IF Main.Errors.InMoldDryingErrors.TopMoldB.HeatingZone[6].PT100_HasWrongPosition THEN 
Topmold_B_heating_Zone_6_PT100_wrong_position.Raise(0); 
END_IF 

IF Main.Errors.InMoldDryingErrors.TopMoldB.HeatingZone[6].PT100_Loose THEN 
Topmold_B_heating_Zone_6_PT100_loose.Raise(0); 
END_IF 

IF Main.Errors.InMoldDryingErrors.TopMoldB.HeatingZone[6].PT100_NotInserted THEN 
Topmold_B_heating_Zone_6_PT100_not_inserted.Raise(0); 
END_IF 

IF Main.Errors.InMoldDryingErrors.TopMoldB.HeatingZone[6].PT100_TempAboveSetpoint THEN 
Topmold_B_heating_Zone_6_Temperature_above_setpoint.Raise(0); 
END_IF 

IF Main.Errors.InMoldDryingErrors.TopMoldB.HeatingZone[6].PT100_TempBelowSetpoint THEN 
Topmold_B_heating_Zone_6_Temperature_below_setpoint.Raise(0); 
END_IF 

IF Main.Errors.InMoldDryingErrors.TopMoldB.HeatingZone[6].PT100_WireBreak THEN 
Topmold_B_heating_Zone_6_PT100_wirebreak.Raise(0); 
END_IF 

IF Main.Errors.InMoldDryingErrors.TopMoldB.HeatingZone[6].Thermal THEN 
Topmold_B_heating_Zone_6_Thermal.Raise(0); 
END_IF 

IF Main.Errors.InMoldDryingErrors.TopMoldB.HeatingZone[6].PT100_TemperatureAboveMaximum THEN 
Topmold_B_heating_zone_6_temperature_above_250_degree_heating_element_switched_off.Raise(0); 
END_IF 

IF Main.Errors.InMoldDryingErrors.TopMoldB.HeatingZone[6].PT100_TemperatureTooHighWarn THEN 
Topmold_B_heating_zone_6_temperature_above_230_degree.Raise(0); 
END_IF 

IF Main.Errors.InMoldDryingErrors.TopMoldB.Hydraulic.BallufError THEN 
Bottom_mold_B_error_on_balluf.Raise(0); 
END_IF 

IF Main.Errors.InMoldDryingErrors.TopMoldB.Hydraulic.IsMovingWithoutActivation THEN 
Bottom_mold_B_is_moving_without_activation.Raise(0); 
END_IF 

IF FALSE THEN 
Top_mold_B_Bot_side_pressure_too_high.Raise(0); 
END_IF 

IF FALSE THEN 
Top_mold_B_Rot_side_pressure_too_high.Raise(0); 
END_IF 

IF Main.Errors.InMoldDryingErrors.BottomMoldB.HeatingZone[1].PT100_ConnectorNotConnected THEN 
Bottom_mold_B_heating_Zone_1_connector_not_connected.Raise(0); 
END_IF 

IF Main.Errors.InMoldDryingErrors.BottomMoldB.HeatingZone[1].PT100_HasWrongPosition THEN 
Bottom_mold_B_heating_Zone_1_PT100_wrong_position.Raise(0); 
END_IF 

IF Main.Errors.InMoldDryingErrors.BottomMoldB.HeatingZone[1].PT100_Loose THEN 
Bottom_mold_B_heating_Zone_1_PT100_loose.Raise(0); 
END_IF 

IF Main.Errors.InMoldDryingErrors.BottomMoldB.HeatingZone[1].PT100_NotInserted THEN 
Bottom_mold_B_heating_Zone_1_PT100_not_inserted.Raise(0); 
END_IF 

IF Main.Errors.InMoldDryingErrors.BottomMoldB.HeatingZone[1].PT100_TempAboveSetpoint THEN 
Bottom_mold_B_heating_Zone_1_Temperature_above_setpoint.Raise(0); 
END_IF 

IF Main.Errors.InMoldDryingErrors.BottomMoldB.HeatingZone[1].PT100_TempBelowSetpoint THEN 
Bottom_mold_B_heating_Zone_1_Temperature_below_setpoint.Raise(0); 
END_IF 

IF Main.Errors.InMoldDryingErrors.BottomMoldB.HeatingZone[1].PT100_WireBreak THEN 
Bottom_mold_B_heating_Zone_1_PT100_wirebreak.Raise(0); 
END_IF 

IF Main.Errors.InMoldDryingErrors.BottomMoldB.HeatingZone[1].Thermal THEN 
Bottom_mold_B_heating_Zone_1_Thermal.Raise(0); 
END_IF 

IF Main.Errors.InMoldDryingErrors.BottomMoldB.HeatingZone[1].PT100_TemperatureAboveMaximum THEN 
Bottom_mold_B_heating_zone_1_temperature_above_250_degree_heating_element_switched_off.Raise(0); 
END_IF 

IF Main.Errors.InMoldDryingErrors.BottomMoldB.HeatingZone[1].PT100_TemperatureTooHighWarn THEN 
Bottom_mold_B_heating_zone_1_temperature_above_230_degree.Raise(0); 
END_IF 

IF Main.Errors.InMoldDryingErrors.BottomMoldB.HeatingZone[2].PT100_ConnectorNotConnected THEN 
Bottom_mold_B_heating_Zone_2_connector_not_connected.Raise(0); 
END_IF 

IF Main.Errors.InMoldDryingErrors.BottomMoldB.HeatingZone[2].PT100_HasWrongPosition THEN 
Bottom_mold_B_heating_Zone_2_PT100_wrong_position.Raise(0); 
END_IF 

IF Main.Errors.InMoldDryingErrors.BottomMoldB.HeatingZone[2].PT100_Loose THEN 
Bottom_mold_B_heating_Zone_2_PT100_loose.Raise(0); 
END_IF 

IF Main.Errors.InMoldDryingErrors.BottomMoldB.HeatingZone[2].PT100_NotInserted THEN 
Bottom_mold_B_heating_Zone_2_PT100_not_inserted.Raise(0); 
END_IF 

IF Main.Errors.InMoldDryingErrors.BottomMoldB.HeatingZone[2].PT100_TempAboveSetpoint THEN 
Bottom_mold_B_heating_Zone_2_Temperature_above_setpoint.Raise(0); 
END_IF 

IF Main.Errors.InMoldDryingErrors.BottomMoldB.HeatingZone[2].PT100_TempBelowSetpoint THEN 
Bottom_mold_B_heating_Zone_2_Temperature_below_setpoint.Raise(0); 
END_IF 

IF Main.Errors.InMoldDryingErrors.BottomMoldB.HeatingZone[2].PT100_WireBreak THEN 
Bottom_mold_B_heating_Zone_2_PT100_wirebreak.Raise(0); 
END_IF 

IF Main.Errors.InMoldDryingErrors.BottomMoldB.HeatingZone[2].Thermal THEN 
Bottom_mold_B_heating_Zone_2_Thermal.Raise(0); 
END_IF 

IF Main.Errors.InMoldDryingErrors.BottomMoldB.HeatingZone[2].PT100_TemperatureAboveMaximum THEN 
Bottom_mold_B_heating_zone_2_temperature_above_250_degree_heating_element_switched_off.Raise(0); 
END_IF 

IF Main.Errors.InMoldDryingErrors.BottomMoldB.HeatingZone[2].PT100_TemperatureTooHighWarn THEN 
Bottom_mold_B_heating_zone_2_temperature_above_230_degree.Raise(0); 
END_IF 

IF Main.Errors.InMoldDryingErrors.BottomMoldB.HeatingZone[3].PT100_ConnectorNotConnected THEN 
Bottom_mold_B_heating_Zone_3_connector_not_connected.Raise(0); 
END_IF 

IF Main.Errors.InMoldDryingErrors.BottomMoldB.HeatingZone[3].PT100_HasWrongPosition THEN 
Bottom_mold_B_heating_Zone_3_PT100_wrong_position.Raise(0); 
END_IF 

IF Main.Errors.InMoldDryingErrors.BottomMoldB.HeatingZone[3].PT100_Loose THEN 
Bottom_mold_B_heating_Zone_3_PT100_loose.Raise(0); 
END_IF 

IF Main.Errors.InMoldDryingErrors.BottomMoldB.HeatingZone[3].PT100_NotInserted THEN 
Bottom_mold_B_heating_Zone_3_PT100_not_inserted.Raise(0); 
END_IF 

IF Main.Errors.InMoldDryingErrors.BottomMoldB.HeatingZone[3].PT100_TempAboveSetpoint THEN 
Bottom_mold_B_heating_Zone_3_Temperature_above_setpoint.Raise(0); 
END_IF 

IF Main.Errors.InMoldDryingErrors.BottomMoldB.HeatingZone[3].PT100_TempBelowSetpoint THEN 
Bottom_mold_B_heating_Zone_3_Temperature_below_setpoint.Raise(0); 
END_IF 

IF Main.Errors.InMoldDryingErrors.BottomMoldB.HeatingZone[3].PT100_WireBreak THEN 
Bottom_mold_B_heating_Zone_3_PT100_wirebreak.Raise(0); 
END_IF 

IF Main.Errors.InMoldDryingErrors.BottomMoldB.HeatingZone[3].Thermal THEN 
Bottom_mold_B_heating_Zone_3_Thermal.Raise(0); 
END_IF 

IF Main.Errors.InMoldDryingErrors.BottomMoldB.HeatingZone[3].PT100_TemperatureAboveMaximum THEN 
Bottom_mold_B_heating_zone_3_temperature_above_250_degree_heating_element_switched_off.Raise(0); 
END_IF 

IF Main.Errors.InMoldDryingErrors.BottomMoldB.HeatingZone[3].PT100_TemperatureTooHighWarn THEN 
Bottom_mold_B_heating_zone_3_temperature_above_230_degree.Raise(0); 
END_IF 

IF Main.Errors.InMoldDryingErrors.BottomMoldB.HeatingZone[4].PT100_ConnectorNotConnected THEN 
Bottom_mold_B_heating_Zone_4_connector_not_connected.Raise(0); 
END_IF 

IF Main.Errors.InMoldDryingErrors.BottomMoldB.HeatingZone[4].PT100_HasWrongPosition THEN 
Bottom_mold_B_heating_Zone_4_PT100_wrong_position.Raise(0); 
END_IF 

IF Main.Errors.InMoldDryingErrors.BottomMoldB.HeatingZone[4].PT100_Loose THEN 
Bottom_mold_B_heating_Zone_4_PT100_loose.Raise(0); 
END_IF 

IF Main.Errors.InMoldDryingErrors.BottomMoldB.HeatingZone[4].PT100_NotInserted THEN 
Bottom_mold_B_heating_Zone_4_PT100_not_inserted.Raise(0); 
END_IF 

IF Main.Errors.InMoldDryingErrors.BottomMoldB.HeatingZone[4].PT100_TempAboveSetpoint THEN 
Bottom_mold_B_heating_Zone_4_Temperature_above_setpoint.Raise(0); 
END_IF 

IF Main.Errors.InMoldDryingErrors.BottomMoldB.HeatingZone[4].PT100_TempBelowSetpoint THEN 
Bottom_mold_B_heating_Zone_4_Temperature_below_setpoint.Raise(0); 
END_IF 

IF Main.Errors.InMoldDryingErrors.BottomMoldB.HeatingZone[4].PT100_WireBreak THEN 
Bottom_mold_B_heating_Zone_4_PT100_wirebreak.Raise(0); 
END_IF 

IF Main.Errors.InMoldDryingErrors.BottomMoldB.HeatingZone[4].Thermal THEN 
Bottom_mold_B_heating_Zone_4_Thermal.Raise(0); 
END_IF 

IF Main.Errors.InMoldDryingErrors.BottomMoldB.HeatingZone[4].PT100_TemperatureAboveMaximum THEN 
Bottom_mold_B_heating_zone_4_temperature_above_250_degree_heating_element_switched_off.Raise(0); 
END_IF 

IF Main.Errors.InMoldDryingErrors.BottomMoldB.HeatingZone[4].PT100_TemperatureTooHighWarn THEN 
Bottom_mold_B_heating_zone_4_temperature_above_230_degree.Raise(0); 
END_IF 

IF Main.Errors.InMoldDryingErrors.BottomMoldB.HeatingZone[5].PT100_ConnectorNotConnected THEN 
Bottom_mold_B_heating_Zone_5_connector_not_connected.Raise(0); 
END_IF 

IF Main.Errors.InMoldDryingErrors.BottomMoldB.HeatingZone[5].PT100_HasWrongPosition THEN 
Bottom_mold_B_heating_Zone_5_PT100_wrong_position.Raise(0); 
END_IF 

IF Main.Errors.InMoldDryingErrors.BottomMoldB.HeatingZone[5].PT100_Loose THEN 
Bottom_mold_B_heating_Zone_5_PT100_loose.Raise(0); 
END_IF 

IF Main.Errors.InMoldDryingErrors.BottomMoldB.HeatingZone[5].PT100_NotInserted THEN 
Bottom_mold_B_heating_Zone_5_PT100_not_inserted.Raise(0); 
END_IF 

IF Main.Errors.InMoldDryingErrors.BottomMoldB.HeatingZone[5].PT100_TempAboveSetpoint THEN 
Bottom_mold_B_heating_Zone_5_Temperature_above_setpoint.Raise(0); 
END_IF 

IF Main.Errors.InMoldDryingErrors.BottomMoldB.HeatingZone[5].PT100_TempBelowSetpoint THEN 
Bottom_mold_B_heating_Zone_5_Temperature_below_setpoint.Raise(0); 
END_IF 

IF Main.Errors.InMoldDryingErrors.BottomMoldB.HeatingZone[5].PT100_WireBreak THEN 
Bottom_mold_B_heating_Zone_5_PT100_wirebreak.Raise(0); 
END_IF 

IF Main.Errors.InMoldDryingErrors.BottomMoldB.HeatingZone[5].Thermal THEN 
Bottom_mold_B_heating_Zone_5_Thermal.Raise(0); 
END_IF 

IF Main.Errors.InMoldDryingErrors.BottomMoldB.HeatingZone[5].PT100_TemperatureAboveMaximum THEN 
Bottom_mold_B_heating_zone_5_temperature_above_250_degree_heating_element_switched_off.Raise(0); 
END_IF 

IF Main.Errors.InMoldDryingErrors.BottomMoldB.HeatingZone[5].PT100_TemperatureTooHighWarn THEN 
Bottom_mold_B_heating_zone_5_temperature_above_230_degree.Raise(0); 
END_IF 

IF Main.Errors.InMoldDryingErrors.BottomMoldB.HeatingZone[6].PT100_ConnectorNotConnected THEN 
Bottom_mold_B_heating_Zone_6_connector_not_connected.Raise(0); 
END_IF 

IF Main.Errors.InMoldDryingErrors.BottomMoldB.HeatingZone[6].PT100_HasWrongPosition THEN 
Bottom_mold_B_heating_Zone_6_PT100_wrong_position.Raise(0); 
END_IF 

IF Main.Errors.InMoldDryingErrors.BottomMoldB.HeatingZone[6].PT100_Loose THEN 
Bottom_mold_B_heating_Zone_6_PT100_loose.Raise(0); 
END_IF 

IF Main.Errors.InMoldDryingErrors.BottomMoldB.HeatingZone[6].PT100_NotInserted THEN 
Bottom_mold_B_heating_Zone_6_PT100_not_inserted.Raise(0); 
END_IF 

IF Main.Errors.InMoldDryingErrors.BottomMoldB.HeatingZone[6].PT100_TempAboveSetpoint THEN 
Bottom_mold_B_heating_Zone_6_Temperature_above_setpoint.Raise(0); 
END_IF 

IF Main.Errors.InMoldDryingErrors.BottomMoldB.HeatingZone[6].PT100_TempBelowSetpoint THEN 
Bottom_mold_B_heating_Zone_6_Temperature_below_setpoint.Raise(0); 
END_IF 

IF Main.Errors.InMoldDryingErrors.BottomMoldB.HeatingZone[6].PT100_WireBreak THEN 
Bottom_mold_B_heating_Zone_6_PT100_wirebreak.Raise(0); 
END_IF 

IF Main.Errors.InMoldDryingErrors.BottomMoldB.HeatingZone[6].Thermal THEN 
Bottom_mold_B_heating_Zone_6_Thermal.Raise(0); 
END_IF 

IF Main.Errors.InMoldDryingErrors.BottomMoldB.HeatingZone[6].PT100_TemperatureAboveMaximum THEN 
Bottom_mold_B_heating_zone_6_temperature_above_250_degree_heating_element_switched_off.Raise(0); 
END_IF 

IF Main.Errors.InMoldDryingErrors.BottomMoldB.HeatingZone[6].PT100_TemperatureTooHighWarn THEN 
Bottom_mold_B_heating_zone_6_temperature_above_230_degree.Raise(0); 
END_IF 

IF Main.Errors.InMoldDryingErrors.BottomMoldA.HorizontalCilinder.Cilinder THEN 
Takeout_unit_A_horizontal_cylinder_error.Raise(0); 
END_IF 

IF Main.Errors.InMoldDryingErrors.BottomMoldA.HorizontalCilinder.CilinderSlow_IN THEN 
Takeout_unit_A_horizontal_cylinder_timeout_in.Raise(0); 
END_IF 

IF Main.Errors.InMoldDryingErrors.BottomMoldA.HorizontalCilinder.CilinderSlow_OUT THEN 
Takeout_unit_A_horizontal_cylinder_timeout_out.Raise(0); 
END_IF 

IF Main.Errors.InMoldDryingErrors.BottomMoldB.HorizontalCilinder.Cilinder THEN 
Takeout_unit_B_horizontal_cylinder_error.Raise(0); 
END_IF 

IF Main.Errors.InMoldDryingErrors.BottomMoldB.HorizontalCilinder.CilinderSlow_IN THEN 
Takeout_unit_B_horizontal_cylinder_timeout_in.Raise(0); 
END_IF 

IF Main.Errors.InMoldDryingErrors.BottomMoldB.HorizontalCilinder.CilinderSlow_OUT THEN 
Takeout_unit_B_horizontal_cylinder_timeout_out.Raise(0); 
END_IF 

IF Main.Errors.InMoldDryingErrors.BottomMoldA.VerticalCilinder.Cilinder THEN 
Takeout_unit_A_vertical_cylinder_error.Raise(0); 
END_IF 

IF Main.Errors.InMoldDryingErrors.BottomMoldA.VerticalCilinder.CilinderSlow_IN THEN 
Takeout_unit_A_vertical_cylinder_timeout_in.Raise(0); 
END_IF 

IF Main.Errors.InMoldDryingErrors.BottomMoldA.VerticalCilinder.CilinderSlow_OUT THEN 
Takeout_unit_A_vertical_cylinder_timeout_out.Raise(0); 
END_IF 

IF Main.Errors.InMoldDryingErrors.BottomMoldB.VerticalCilinder.Cilinder THEN 
Takeout_unit_B_vertical_cylinder_error.Raise(0); 
END_IF 

IF Main.Errors.InMoldDryingErrors.BottomMoldB.VerticalCilinder.CilinderSlow_IN THEN 
Takeout_unit_B_vertical_cylinder_timeout_in.Raise(0); 
END_IF 

IF Main.Errors.InMoldDryingErrors.BottomMoldB.VerticalCilinder.CilinderSlow_OUT THEN 
Takeout_unit_B_vertical_cylinder_timeout_out.Raise(0); 
END_IF 

IF Main.Errors.InMoldDryingErrors.BottomMoldA.VacuumSection[1] THEN 
Takeout_unit_A_error_on_vacuum_section_1.Raise(0); 
END_IF 

IF Main.Errors.InMoldDryingErrors.BottomMoldA.VacuumSection[2] THEN 
Takeout_unit_A_error_on_vacuum_section_2.Raise(0); 
END_IF 

IF Main.Errors.InMoldDryingErrors.BottomMoldA.VacuumSection[3] THEN 
Takeout_unit_A_error_on_vacuum_section_3.Raise(0); 
END_IF 

IF Main.Errors.InMoldDryingErrors.BottomMoldA.VacuumSection[4] THEN 
Takeout_unit_A_error_on_vacuum_section_4.Raise(0); 
END_IF 

IF Main.Errors.InMoldDryingErrors.BottomMoldB.VacuumSection[1] THEN 
Takeout_unit_B_error_on_vacuum_section_1.Raise(0); 
END_IF 

IF Main.Errors.InMoldDryingErrors.BottomMoldB.VacuumSection[2] THEN 
Takeout_unit_B_error_on_vacuum_section_2.Raise(0); 
END_IF 

IF Main.Errors.InMoldDryingErrors.BottomMoldB.VacuumSection[3] THEN 
Takeout_unit_B_error_on_vacuum_section_3.Raise(0); 
END_IF 

IF Main.Errors.InMoldDryingErrors.BottomMoldB.VacuumSection[4] THEN 
Takeout_unit_B_error_on_vacuum_section_4.Raise(0); 
END_IF 

IF Main.Errors.InMoldDryingErrors.ProductForming.HydraulicPump.Maintenance THEN 
Machine_pond_hydraulic_pump_maintenance_switch.Raise(0); 
END_IF 

IF Main.Errors.InMoldDryingErrors.ProductForming.HydraulicPump.Thermal THEN 
Machine_pond_hydraulic_pump_thermal_error.Raise(0); 
END_IF 

IF Main.Errors.InMoldDryingErrors.ProductForming.MachinePond.FeedingPulp.Cilinder THEN 
Machine_oond_pulp_feeding_cylinder_error.Raise(0); 
END_IF 

IF Main.Errors.InMoldDryingErrors.ProductForming.MachinePond.FeedingPulp.CilinderSlow_IN THEN 
Machine_pond_pulp_feeding_cylinder_timeout_in.Raise(0); 
END_IF 

IF Main.Errors.InMoldDryingErrors.ProductForming.MachinePond.FeedingPulp.CilinderSlow_OUT THEN 
Machine_pond_pulp_feeding_cylinder_timeout_out.Raise(0); 
END_IF 

IF Main.Errors.InMoldDryingErrors.TransferMold.HydraulicCilinder.BallufError THEN 
Transfermold_error_on_balluf.Raise(0); 
END_IF 

IF Main.Errors.InMoldDryingErrors.TransferMold.HydraulicCilinder.IsMovingWithoutActivation THEN 
Transfermold_is_moving_without_activation.Raise(0); 
END_IF 

IF Main.Errors.InMoldDryingErrors.RH_BotMoldAToCoolForTrMDown THEN 
RHSR_Bottommold_A_too_cool_for_transfermold_to_come_down.Raise(0); 
END_IF 

IF Main.Errors.InMoldDryingErrors.RH_BotMoldBToCoolForTrMDown THEN 
RHSR_Bottommold_B_too_cool_for_transfermold_to_come_down.Raise(0); 
END_IF 

IF Main.Errors.ProductHandlingErrors.Gantry_A.Collision THEN 
Gantry_A_collision_detected.Raise(0); 
END_IF 

IF Main.Errors.ProductHandlingErrors.Gantry_A.EndLimitHorBack THEN 
Gantry_A_Horizontal_limit_endswitch_backside.Raise(0); 
END_IF 

IF Main.Errors.ProductHandlingErrors.Gantry_A.EndLimitHorFront THEN 
Gantry_A_Horizontal_limit_endswitch_frontside.Raise(0); 
END_IF 

IF Main.Errors.ProductHandlingErrors.Gantry_A.EndLimitVertDown THEN 
Gantry_A_vertical_limit_endswitch_down.Raise(0); 
END_IF 

IF Main.Errors.ProductHandlingErrors.Gantry_A.EndLimitVertUp THEN 
Gantry_A_vertical_limit_endswitch_up.Raise(0); 
END_IF 

IF Main.Errors.ProductHandlingErrors.Gantry_A.HorizontalNCAxisError.exDriveAbsoluut THEN 
Gantry_A_Horizontal_Drive_absoluut_error.Raise(0); 
END_IF 

IF Main.Errors.ProductHandlingErrors.Gantry_A.HorizontalNCAxisError.exDriveJog THEN 
Gantry_A_Horizontal_Drive_Jog_error.Raise(0); 
END_IF 

IF Main.Errors.ProductHandlingErrors.Gantry_A.HorizontalNCAxisError.exDrivePower THEN 
Gantry_A_Horizontal_Drive_power_error.Raise(0); 
END_IF 

IF Main.Errors.ProductHandlingErrors.Gantry_A.HorizontalNCAxisError.exDriveReset THEN 
Gantry_A_Horizontal_Drive_reset.Raise(0); 
END_IF 

IF Main.Errors.ProductHandlingErrors.Gantry_A.HorizontalNCAxisError.exDriveStatus THEN 
Gantry_A_Horizontal_Drive_status.Raise(0); 
END_IF 

IF Main.Errors.ProductHandlingErrors.Gantry_A.HorizontalNCAxisError.exDriveStop THEN 
Gantry_A_Horizontal_Drive_stop_error.Raise(0); 
END_IF 

IF Main.Errors.ProductHandlingErrors.Gantry_A.HorizontalNCAxisError.exDriveVelocity THEN 
Gantry_A_Horizontal_Drive_velocity_error.Raise(0); 
END_IF 

IF Main.Errors.ProductHandlingErrors.Gantry_A.HorizontalNCAxisError.exHome THEN 
Gantry_A_Horizontal_Drive_home_error.Raise(0); 
END_IF 

IF Main.Errors.ProductHandlingErrors.Gantry_A.HorizontalNCAxisError.exLagError THEN 
Gantry_A_Horizontal_Drive_lag_error.Raise(0); 
END_IF 

IF Main.Errors.ProductHandlingErrors.Gantry_A.HorizontalNCAxisError.exReadParameter THEN 
Gantry_A_Horizontal_Drive_read_parameter_error.Raise(0); 
END_IF 

IF Main.Errors.ProductHandlingErrors.Gantry_A.HorizontalNCAxisError.exWriteParameter THEN 
Gantry_A_Horizontal_Drive_write_parameter_error.Raise(0); 
END_IF 

IF Main.Errors.ProductHandlingErrors.Gantry_B.Collision THEN 
Gantry_B_collision_detected.Raise(0); 
END_IF 

IF Main.Errors.ProductHandlingErrors.Gantry_B.EndLimitHorBack THEN 
Gantry_B_horizontal_limit_endswitch_backside.Raise(0); 
END_IF 

IF Main.Errors.ProductHandlingErrors.Gantry_B.EndLimitHorFront THEN 
Gantry_B_horizontal_limit_endswitch_frontside.Raise(0); 
END_IF 

IF Main.Errors.ProductHandlingErrors.Gantry_B.EndLimitVertDown THEN 
Gantry_B_vertical_limit_endswitch_down.Raise(0); 
END_IF 

IF Main.Errors.ProductHandlingErrors.Gantry_B.EndLimitVertUp THEN 
Gantry_B_vertical_limit_endswitch_up.Raise(0); 
END_IF 

IF Main.Errors.ProductHandlingErrors.Gantry_B.HorizontalNCAxisError.exDriveAbsoluut THEN 
Gantry_B_Horizontal_Drive_absoluut_error.Raise(0); 
END_IF 

IF Main.Errors.ProductHandlingErrors.Gantry_B.HorizontalNCAxisError.exDriveJog THEN 
Gantry_B_Horizontal_Drive_Jog_error.Raise(0); 
END_IF 

IF Main.Errors.ProductHandlingErrors.Gantry_B.HorizontalNCAxisError.exDrivePower THEN 
Gantry_B_Horizontal_Drive_power_error.Raise(0); 
END_IF 

IF Main.Errors.ProductHandlingErrors.Gantry_B.HorizontalNCAxisError.exDriveReset THEN 
Gantry_B_Horizontal_Drive_reset.Raise(0); 
END_IF 

IF Main.Errors.ProductHandlingErrors.Gantry_B.HorizontalNCAxisError.exDriveStatus THEN 
Gantry_B_Horizontal_Drive_status.Raise(0); 
END_IF 

IF Main.Errors.ProductHandlingErrors.Gantry_B.HorizontalNCAxisError.exDriveStop THEN 
Gantry_B_Horizontal_Drive_stop_error.Raise(0); 
END_IF 

IF Main.Errors.ProductHandlingErrors.Gantry_B.HorizontalNCAxisError.exDriveVelocity THEN 
Gantry_B_Horizontal_Drive_velocity_error.Raise(0); 
END_IF 

IF Main.Errors.ProductHandlingErrors.Gantry_B.HorizontalNCAxisError.exHome THEN 
Gantry_B_Horizontal_Drive_home_error.Raise(0); 
END_IF 

IF Main.Errors.ProductHandlingErrors.Gantry_B.HorizontalNCAxisError.exLagError THEN 
Gantry_B_Horizontal_Drive_lag_error.Raise(0); 
END_IF 

IF Main.Errors.ProductHandlingErrors.Gantry_B.HorizontalNCAxisError.exReadParameter THEN 
Gantry_B_Horizontal_Drive_read_parameter_error.Raise(0); 
END_IF 

IF Main.Errors.ProductHandlingErrors.Gantry_B.HorizontalNCAxisError.exWriteParameter THEN 
Gantry_B_Horizontal_Drive_write_parameter_error.Raise(0); 
END_IF 

IF Main.Errors.ProductHandlingErrors.RH_HorMovingVertNotAtTranspPos_A THEN 
RHSR_product_handling_gantry_A_is_moving_horizotal_while_vertical_not_on_position.Raise(0); 
END_IF 

IF Main.Errors.ProductHandlingErrors.RH_HorMovingVertNotAtTranspPos_B THEN 
RHSR_product_handling_gantry_B_is_moving_horizotal_while_vertical_not_on_position.Raise(0); 
END_IF 

IF Main.Errors.ProductHandlingErrors.RH_VertMovingHorNotInPos_A THEN 
RHSR_product_handling_gantry_A_is_moving_vertical_while_horizontal_not_on_position.Raise(0); 
END_IF 

IF Main.Errors.ProductHandlingErrors.RH_VertMovingHorNotInPos_B THEN 
RHSR_product_handling_gantry_B_is_moving_vertical_while_horizontal_not_on_position.Raise(0); 
END_IF 

IF Main.Errors.InMoldDryingErrors.ProductForming.SprayBar.NCAxisError.exDriveAbsoluut THEN 
Spraybar_Drive_absoluut_error.Raise(0); 
END_IF 

IF Main.Errors.InMoldDryingErrors.ProductForming.SprayBar.NCAxisError.exDriveJog THEN 
Spraybar_Drive_Jog_error.Raise(0); 
END_IF 

IF Main.Errors.InMoldDryingErrors.ProductForming.SprayBar.NCAxisError.exDrivePower THEN 
Spraybar_Drive_power_error.Raise(0); 
END_IF 

IF Main.Errors.InMoldDryingErrors.ProductForming.SprayBar.NCAxisError.exDriveReset THEN 
Spraybar_Drive_reset.Raise(0); 
END_IF 

IF Main.Errors.InMoldDryingErrors.ProductForming.SprayBar.NCAxisError.exDriveStatus THEN 
Spraybar_Drive_status.Raise(0); 
END_IF 

IF Main.Errors.InMoldDryingErrors.ProductForming.SprayBar.NCAxisError.exDriveStop THEN 
Spraybar_Drive_stop_error.Raise(0); 
END_IF 

IF Main.Errors.InMoldDryingErrors.ProductForming.SprayBar.NCAxisError.exDriveVelocity THEN 
Spraybar_Drive_velocity_error.Raise(0); 
END_IF 

IF Main.Errors.InMoldDryingErrors.ProductForming.SprayBar.NCAxisError.exHome THEN 
Spraybar_Drive_home_error.Raise(0); 
END_IF 

IF Main.Errors.InMoldDryingErrors.ProductForming.SprayBar.NCAxisError.exLagError THEN 
Spraybar_Drive_lag_error.Raise(0); 
END_IF 

IF Main.Errors.InMoldDryingErrors.ProductForming.SprayBar.NCAxisError.exReadParameter THEN 
Spraybar_Drive_read_parameter_error.Raise(0); 
END_IF 

IF Main.Errors.InMoldDryingErrors.ProductForming.SprayBar.NCAxisError.exWriteParameter THEN 
Spraybar_Drive_write_parameter_error.Raise(0); 
END_IF 

IF Main.Errors.ProductHandlingErrors.Gantry_A.ProductLost[1] THEN 
Gantry_A_product_lost_section_1.Raise(0); 
END_IF 

IF Main.Errors.ProductHandlingErrors.Gantry_A.ProductLost[2] THEN 
Gantry_A_product_lost_section_2.Raise(0); 
END_IF 

IF Main.Errors.ProductHandlingErrors.Gantry_A.ProductLost[3] THEN 
Gantry_A_product_lost_section_3.Raise(0); 
END_IF 

IF Main.Errors.ProductHandlingErrors.Gantry_A.ProductLost[4] THEN 
Gantry_A_product_lost_section_4.Raise(0); 
END_IF 

IF Main.Errors.ProductHandlingErrors.Gantry_A.ProductLost[5] THEN 
Gantry_A_product_lost_section_5.Raise(0); 
END_IF 

IF Main.Errors.ProductHandlingErrors.Gantry_A.ProductLost[6] THEN 
Gantry_A_product_lost_section_6.Raise(0); 
END_IF 

IF Main.Errors.ProductHandlingErrors.Gantry_B.ProductLost[1] THEN 
Gantry_B_product_lost_section_1.Raise(0); 
END_IF 

IF Main.Errors.ProductHandlingErrors.Gantry_B.ProductLost[2] THEN 
Gantry_B_product_lost_section_2.Raise(0); 
END_IF 

IF Main.Errors.ProductHandlingErrors.Gantry_B.ProductLost[3] THEN 
Gantry_B_product_lost_section_3.Raise(0); 
END_IF 

IF Main.Errors.ProductHandlingErrors.Gantry_B.ProductLost[4] THEN 
Gantry_B_product_lost_section_4.Raise(0); 
END_IF 

IF Main.Errors.ProductHandlingErrors.Gantry_B.ProductLost[5] THEN 
Gantry_B_product_lost_section_5.Raise(0); 
END_IF 

IF Main.Errors.ProductHandlingErrors.Gantry_B.ProductLost[6] THEN 
Gantry_B_product_lost_section_6.Raise(0); 
END_IF 

IF Main.Errors.InMoldDryingErrors.ProductForming.SprayBar.PositionAtFrontError THEN 
Spraybar_not_in_front_rest_position.Raise(0); 
END_IF 

IF Main.Errors.InMoldDryingErrors.ProductForming.SprayBar.PositionAtBackError THEN 
Spraybar_not_in_back_rest_position.Raise(0); 
END_IF 

IF MAIN.EtherCatDiag.EtherCATLinkError THEN 
Ethercat_diagnosed_a_link_error.Raise(0); 
END_IF 

IF MAIN.EtherCatDiag.EtherCATSlaveMissing THEN 
Ethercat_diagnosed_that_a_slave_is_missing.Raise(0); 
END_IF 

IF MAIN.EtherCatDiag.EtherCATOPmode THEN 
Ethercat_diagnosed_a_non_OP_state.Raise(0); 
END_IF 

IF MAIN.EtherCatDiag.EtherCATResetNeeded THEN 
Ethercat_diagnosed_that_a_ethercat_reset_is_needed.Raise(0); 
END_IF 

IF Main.Errors.InMoldDryingErrors.TopMoldA.Hydraulic.SafePositionValveNotReached THEN 
TopMold_A_Safe_position_not_reached.Raise(0); 
END_IF 

IF Main.Errors.InMoldDryingErrors.TopMoldB.Hydraulic.SafePositionValveNotReached THEN 
TopMold_B_Safe_position_not_reached.Raise(0); 
END_IF 

IF Main.Errors.InMoldDryingErrors.TransferMold.HydraulicCilinder.SafePositionValveNotReached THEN 
Transfermold_Safe_position_not_reached.Raise(0); 
END_IF 

IF Main.Errors.InMoldDryingErrors.TempDeviationToHighA[1] THEN 
Difference_in_temperature_too_high_top_bottommold_A_zone_1.Raise(0); 
END_IF 

IF Main.Errors.InMoldDryingErrors.TempDeviationToHighA[2] THEN 
Difference_in_temperature_too_high_top_bottommold_A_zone_2.Raise(0); 
END_IF 

IF Main.Errors.InMoldDryingErrors.TempDeviationToHighA[3] THEN 
Difference_in_temperature_too_high_top_bottommold_A_zone_3.Raise(0); 
END_IF 

IF Main.Errors.InMoldDryingErrors.TempDeviationToHighA[4] THEN 
Difference_in_temperature_too_high_top_bottommold_A_zone_4.Raise(0); 
END_IF 

IF Main.Errors.InMoldDryingErrors.TempDeviationToHighA[5] THEN 
Difference_in_temperature_too_high_top_bottommold_A_zone_5.Raise(0); 
END_IF 

IF Main.Errors.InMoldDryingErrors.TempDeviationToHighA[6] THEN 
Difference_in_temperature_too_high_top_bottommold_A_zone_6.Raise(0); 
END_IF 

IF Main.Errors.InMoldDryingErrors.TempDeviationToHighB[1] THEN 
Difference_in_temperature_too_high_top_bottommold_B_zone_1.Raise(0); 
END_IF 

IF Main.Errors.InMoldDryingErrors.TempDeviationToHighB[2] THEN 
Difference_in_temperature_too_high_top_bottommold_B_zone_2.Raise(0); 
END_IF 

IF Main.Errors.InMoldDryingErrors.TempDeviationToHighB[3] THEN 
Difference_in_temperature_too_high_top_bottommold_B_zone_3.Raise(0); 
END_IF 

IF Main.Errors.InMoldDryingErrors.TempDeviationToHighB[4] THEN 
Difference_in_temperature_too_high_top_bottommold_B_zone_4.Raise(0); 
END_IF 

IF Main.Errors.InMoldDryingErrors.TempDeviationToHighB[5] THEN 
Difference_in_temperature_too_high_top_bottommold_B_zone_5.Raise(0); 
END_IF 

IF Main.Errors.InMoldDryingErrors.TempDeviationToHighB[6] THEN 
Difference_in_temperature_too_high_top_bottommold_B_zone_6.Raise(0); 
END_IF 

IF Main.Errors.ProductHandlingErrors.Gantry_A.VerticalNCAxisError.exDriveAbsoluut THEN 
Gantry_A_Vertical_Drive_absoluut_error.Raise(0); 
END_IF 

IF Main.Errors.ProductHandlingErrors.Gantry_A.VerticalNCAxisError.exDriveJog THEN 
Gantry_A_Vertical_Drive_Jog_error.Raise(0); 
END_IF 

IF Main.Errors.ProductHandlingErrors.Gantry_A.VerticalNCAxisError.exDrivePower THEN 
Gantry_A_Vertical_Drive_power_error.Raise(0); 
END_IF 

IF Main.Errors.ProductHandlingErrors.Gantry_A.VerticalNCAxisError.exDriveReset THEN 
Gantry_A_Vertical_Drive_reset.Raise(0); 
END_IF 

IF Main.Errors.ProductHandlingErrors.Gantry_A.VerticalNCAxisError.exDriveStatus THEN 
Gantry_A_Vertical_Drive_status.Raise(0); 
END_IF 

IF Main.Errors.ProductHandlingErrors.Gantry_A.VerticalNCAxisError.exDriveStop THEN 
Gantry_A_Vertical_Drive_stop_error.Raise(0); 
END_IF 

IF Main.Errors.ProductHandlingErrors.Gantry_A.VerticalNCAxisError.exDriveVelocity THEN 
Gantry_A_Vertical_Drive_velocity_error.Raise(0); 
END_IF 

IF Main.Errors.ProductHandlingErrors.Gantry_A.VerticalNCAxisError.exHome THEN 
Gantry_A_Vertical_Drive_home_error.Raise(0); 
END_IF 

IF Main.Errors.ProductHandlingErrors.Gantry_A.VerticalNCAxisError.exLagError THEN 
Gantry_A_Vertical_Drive_lag_error.Raise(0); 
END_IF 

IF Main.Errors.ProductHandlingErrors.Gantry_A.VerticalNCAxisError.exReadParameter THEN 
Gantry_A_Vertical_Drive_read_parameter_error.Raise(0); 
END_IF 

IF Main.Errors.ProductHandlingErrors.Gantry_A.VerticalNCAxisError.exWriteParameter THEN 
Gantry_A_Vertical_Drive_write_parameter_error.Raise(0); 
END_IF 

IF Main.Errors.ProductHandlingErrors.Gantry_B.VerticalNCAxisError.exDriveAbsoluut THEN 
Gantry_B_Vertical_Drive_absoluut_error.Raise(0); 
END_IF 

IF Main.Errors.ProductHandlingErrors.Gantry_B.VerticalNCAxisError.exDriveJog THEN 
Gantry_B_Vertical_Drive_Jog_error.Raise(0); 
END_IF 

IF Main.Errors.ProductHandlingErrors.Gantry_B.VerticalNCAxisError.exDrivePower THEN 
Gantry_B_Vertical_Drive_power_error.Raise(0); 
END_IF 

IF Main.Errors.ProductHandlingErrors.Gantry_B.VerticalNCAxisError.exDriveReset THEN 
Gantry_B_Vertical_Drive_reset.Raise(0); 
END_IF 

IF Main.Errors.ProductHandlingErrors.Gantry_B.VerticalNCAxisError.exDriveStatus THEN 
Gantry_B_Vertical_Drive_status.Raise(0); 
END_IF 

IF Main.Errors.ProductHandlingErrors.Gantry_B.VerticalNCAxisError.exDriveStop THEN 
Gantry_B_Vertical_Drive_stop_error.Raise(0); 
END_IF 

IF Main.Errors.ProductHandlingErrors.Gantry_B.VerticalNCAxisError.exDriveVelocity THEN 
Gantry_B_Vertical_Drive_velocity_error.Raise(0); 
END_IF 

IF Main.Errors.ProductHandlingErrors.Gantry_B.VerticalNCAxisError.exHome THEN 
Gantry_B_Vertical_Drive_home_error.Raise(0); 
END_IF 

IF Main.Errors.ProductHandlingErrors.Gantry_B.VerticalNCAxisError.exLagError THEN 
Gantry_B_Vertical_Drive_lag_error.Raise(0); 
END_IF 

IF Main.Errors.ProductHandlingErrors.Gantry_B.VerticalNCAxisError.exReadParameter THEN 
Gantry_B_Vertical_Drive_read_parameter_error.Raise(0); 
END_IF 

IF Main.Errors.ProductHandlingErrors.Gantry_B.VerticalNCAxisError.exWriteParameter THEN 
Gantry_B_Vertical_Drive_write_parameter_error.Raise(0); 
END_IF 

IF Main.Errors.InMoldDryingErrors.BottomMoldB.HorizontalAxis.exDriveAbsoluut THEN 
Bottommold_B_Horizontal_Drive_absoluut_error.Raise(0); 
END_IF 

IF Main.Errors.InMoldDryingErrors.BottomMoldB.HorizontalAxis.exDriveJog THEN 
Bottommold_B_Horizontal_Drive_Jog_error.Raise(0); 
END_IF 

IF Main.Errors.InMoldDryingErrors.BottomMoldB.HorizontalAxis.exDrivePower THEN 
Bottommold_B_Horizontal_Drive_power_error.Raise(0); 
END_IF 

IF Main.Errors.InMoldDryingErrors.BottomMoldB.HorizontalAxis.exDriveReset THEN 
Bottommold_B_Horizontal_Drive_reset.Raise(0); 
END_IF 

IF Main.Errors.InMoldDryingErrors.BottomMoldB.HorizontalAxis.exDriveStatus THEN 
Bottommold_B_Horizontal_Drive_status.Raise(0); 
END_IF 

IF Main.Errors.InMoldDryingErrors.BottomMoldB.HorizontalAxis.exDriveStop THEN 
Bottommold_B_Horizontal_Drive_stop_error.Raise(0); 
END_IF 

IF Main.Errors.InMoldDryingErrors.BottomMoldB.HorizontalAxis.exDriveVelocity THEN 
Bottommold_B_Horizontal_Drive_velocity_error.Raise(0); 
END_IF 

IF Main.Errors.InMoldDryingErrors.BottomMoldB.HorizontalAxis.exHome THEN 
Bottommold_B_Horizontal_Drive_home_error.Raise(0); 
END_IF 

IF Main.Errors.InMoldDryingErrors.BottomMoldB.HorizontalAxis.exLagError THEN 
Bottommold_B_Horizontal_Drive_lag_error.Raise(0); 
END_IF 

IF Main.Errors.InMoldDryingErrors.BottomMoldB.HorizontalAxis.exReadParameter THEN 
Bottommold_B_Horizontal_Drive_read_parameter_error.Raise(0); 
END_IF 

IF Main.Errors.InMoldDryingErrors.BottomMoldB.HorizontalAxis.exWriteParameter THEN 
Bottommold_B_Horizontal_Drive_write_parameter_error.Raise(0); 
END_IF 

IF Main.Errors.InMoldDryingErrors.BottomMoldA.HorizontalAxis.exDriveAbsoluut THEN 
Bottommold_A_Horizontal_Drive_absoluut_error.Raise(0); 
END_IF 

IF Main.Errors.InMoldDryingErrors.BottomMoldA.HorizontalAxis.exDriveJog THEN 
Bottommold_A_Horizontal_Drive_Jog_error.Raise(0); 
END_IF 

IF Main.Errors.InMoldDryingErrors.BottomMoldA.HorizontalAxis.exDrivePower THEN 
Bottommold_A_Horizontal_Drive_power_error.Raise(0); 
END_IF 

IF Main.Errors.InMoldDryingErrors.BottomMoldA.HorizontalAxis.exDriveReset THEN 
Bottommold_A_Horizontal_Drive_reset.Raise(0); 
END_IF 

IF Main.Errors.InMoldDryingErrors.BottomMoldA.HorizontalAxis.exDriveStatus THEN 
Bottommold_A_Horizontal_Drive_status.Raise(0); 
END_IF 

IF Main.Errors.InMoldDryingErrors.BottomMoldA.HorizontalAxis.exDriveStop THEN 
Bottommold_A_Horizontal_Drive_stop_error.Raise(0); 
END_IF 

IF Main.Errors.InMoldDryingErrors.BottomMoldA.HorizontalAxis.exDriveVelocity THEN 
Bottommold_A_Horizontal_Drive_velocity_error.Raise(0); 
END_IF 

IF Main.Errors.InMoldDryingErrors.BottomMoldA.HorizontalAxis.exHome THEN 
Bottommold_A_Horizontal_Drive_home_error.Raise(0); 
END_IF 

IF Main.Errors.InMoldDryingErrors.BottomMoldA.HorizontalAxis.exLagError THEN 
Bottommold_A_Horizontal_Drive_lag_error.Raise(0); 
END_IF 

IF Main.Errors.InMoldDryingErrors.BottomMoldA.HorizontalAxis.exReadParameter THEN 
Bottommold_A_Horizontal_Drive_read_parameter_error.Raise(0); 
END_IF 

IF Main.Errors.InMoldDryingErrors.BottomMoldA.HorizontalAxis.exWriteParameter THEN 
Bottommold_A_Horizontal_Drive_write_parameter_error.Raise(0); 
END_IF
END_ACTION

END_PROGRAM

// ---- POUs/InMoldDrying/BottomMold/FB_BottomMold.TcPOU
FUNCTION_BLOCK FB_BottomMold
VAR CONSTANT
	sCycleStateTextDef: ARRAY[0..10]  OF STRING :=	
		['State 0: Wait for Start',
		'State 1: Wait for transfer / drying ready to move in',
		'State 2: Move bottom mold in',
		'State 3: Move take out vertical up',
		'State 4: Move take out vertical down',
		'State 5: Wait for transfer is down, and vacuum on',
		'State 6: Wait for transfer is up and ready',
		'State 7: Move bottommold out, take out horizontal in',
		'State 8: Awaiting finnished product picked up by Gantry',
		'State 9: Move take out in',
		'State 10: Error'];
	
	tCycleStateTimeouts: ARRAY[0..10] OF TIME := 
		[T#10S,T#10S,T#10S,T#10S,T#10S,T#10S,T#10S,T#10S,T#10S,T#10S,
		T#10S];

	sInitStateTextDef: ARRAY[0..10] OF STRING :=
		['State 0: Wait for Init start',
		'State 1: Move vertical air cylinder down',
		'State 2: Move bottommold out',
		'State 3; Move horizontal air cylinder out',
		'State 4: ',
		'State 5: ',
		'State 6: ',
		'State 7: ',
		'State 8: ',
		'State 9: ',
		'State 10: Stop init state'];

	tInitStateTimeouts: ARRAY[0..10] OF TIME := 
		[T#10S,T#10S,T#10S,T#10S,T#10S,T#10S,T#10S,T#10S,T#10S,T#10S
		,T#10S];
END_VAR

VAR_INPUT
	mxResetCycleState				: BOOL;
	mxResetInitState				: BOOL;
	mxForceInit						: BOOL; (*Reset Calibration Flag*)
	mxReset							: BOOL;	(*Reset Error*)
	mxEmergency						: BOOL;
	mxDoorsOpened					: BOOL;
	mxAutoMode						: BOOL; (* TRUE = Automode *)
	mxEmptyMachine					: BOOL;
	mxEnableHeating					: BOOL;
	


	mxGantryPickedUpProduct			: BOOL;

	mxTransferIsAtTransferPos		: BOOL;
	TransferPosA					: REAL;
	TransferPosB					: REAL;
	ContinueWithA					: BOOL;
	ContinueWithB					: BOOL;

	mxProductReadyForGantry			: BOOL; (* Signal to gantry, take out product *)

	mxVacuumOn						: BOOL;
	mxProductOnTopMold				: BOOL;

	ActualPositionTransfermold		: REAL;
	RHSR_Blocked 					: BOOL;
	
	(*Signals*)
	SgMoveIn						: BOOL; (* Signal from transfer mold *)
	sgMoveOut						: BOOL; (* Signal from transfer mold *)
	SgBottomIsIn					: BOOL; (* Signal to transfer *)
	SgBottomIsOut					: BOOL; (* Signal to TopMold, move down to dry *)
	SgMoldsAreClosed				: BOOL; (* Signal that indicates that the topmold is closed on the bottommold.*)
END_VAR
VAR_IN_OUT
	MachParameters					: ST_BottomMoldMachPar;
	SysParameters					: ST_BottomMoldSysPar;
	ProdParameters					: ST_BottomMoldProdPar;
END_VAR
VAR_OUTPUT
(*Errors*)
	Errors							: ST_BottomMoldErrors;
	mxErrorInit						: BOOL;		(* Error, stop immediately. Initialisation neccesary *)
	mxErrorStopinPos				: BOOL;		(* Error, stop in position. Only reset neccesary *)

(* State vars *)
	mxCycleBusy						: BOOL;
	mxInitBusy						: BOOL;
	
(* Vars *)
	mxInitialized					: BOOL;
	mxReadyForTransfer				: BOOL;
		
	mxProductReadyAtTakeOut			: BOOL; (* Signal to gantry, take out product *)
	mxTakeoutIsMovingUp				: BOOL;
	
	mxCilIsMovingIn					: BOOL;
	mxCilIsMovingOut				: BOOL;
	mxCilIsIn						: BOOL;
	mxCilIsOut						: BOOL;	
	mxHorCilIsIn					: BOOL;
	mxHorCilIsOut					: BOOL;
	mxVertCilIsIn					: BOOL;
	mxVertCilIsOut					: BOOL;
	
	ActualPosition					: REAL;
END_VAR
VAR
(* State vars *)
	miCycleState					: INT :=0;
	miCycleOldstate					: INT :=0;
	mxCycleTransitionState			: BOOL := FALSE;
	sCycleStateText					: STRING;
	exCycleTimeOut					: BOOL;		(* Timeout for the whole programcycle *)
	CycleTimeout					: TON;
	CycleTimeOutUpFlank				: R_TRIG;
	mxCycleTimeoutEnable			: BOOL;
	CycleTime						: REAL;
	mxCycleHasError					: BOOL;
	miStopState						: INT;
	mxStartCycle					: BOOL;
	mxStopCycle						: BOOL;
	mxStopDirect					: BOOL;
	
	miInitState						: INT	:=0;
	miInitOldstate					: INT	:=0;
	mxInitTransitionState			: BOOL	:= FALSE;
	sInitStateText					: STRING;
	exInitTimeOut					: BOOL;		(* Timeout for the whole programcycle *)
	InitTimeout						: TON;
	InitTimeOutUpFlank				: R_TRIG;
	mxInitTimeoutEnable				: BOOL;
	InitTime						: REAL;
	mxInitHasError					: BOOL;
	mxStartInit						: BOOL;
	mxStopInit						: BOOL;
	

(* Objects *)
	HorizontalCilinder				: FB_BiValve2Fdbck;
	VerticalCilinder				: FB_BiValve2Fdbck;
	HorizontalAxis					: FB_NcAxis;
	VacuumTakeout					: ARRAY [1..6] OF FB_MonoValveNoFdbck;	(* IMD-V *)		
	VacuumSensor					AT %I* : ARRAY [1..6] OF BOOL;
	
	HeatingZone						: ARRAY [1..6] OF FB_Heatingzone;
	

	Vacuum							: FB_MonoValveNoFdbck;	(* IMD-V *)		
	
(* Vars *)
	T_TakeOutTime					: TON;
	T_VacSectionDelay				: ARRAY [1..GVL.MaxNrOfVacSectTakeOutUnit] OF TON;
	SR_ErrorNoVacAtSection			: ARRAY [1..GVL.MaxNrOfVacSectTakeOutUnit] OF SR;
	mxSwitchVacuumOn				: BOOL;
	miVacSection					: INT;
	T_VCilinderMoveOut				: TON;
	T_VCilinderMoveIn				: TON;
	
	RT_GantryPickedUpProduct 		: R_TRIG;
	//T_VacuumDelayedOff				: TON;
	FT_SwitchVacuumOff				: F_TRIG;
	T_TestBigBang					: TON;
	mxFirstCycle					: BOOL;
	
	mrAxisIsMoving					: BOOL;
	mrAxisActPos					: LREAL;
	RT_MoveToGreasingPosition: R_TRIG;
	mxHMI_MoveToGreasingPos: BOOL;
	T_VacuumBottomMoldClosed: TON;
	RT_VacuumBottomMoldClosed: R_TRIG;
END_VAR

Error();
Init();
Cycle();
Objects();

ActualPosition := LREAL_TO_REAL(HorizontalAxis.ActPosition);

mxCilIsIn := ((ActualPosition < (MachParameters.PositionInStop + 1)) AND (ActualPosition > (MachParameters.PositionInStop - 1))); 
mxCilIsOut := ((ActualPosition < (MachParameters.PositionOutStop + 1)) AND (ActualPosition > (MachParameters.PositionOutStop - 1))); 

// Move to Greasing Position
IF mxHMI_MoveToGreasingPos AND NOT mxCycleBusy AND NOT mxAutoMode THEN
	IF HorizontalAxis.M_MoveAbsolute(MachParameters.GreasingVelocity, MachParameters.GreasingPosition) THEN
		mxHMI_MoveToGreasingPos := FALSE;
	END_IF	
END_IF

ACTION Cycle:
(*StateChange (Transition)  Signalgeneration*)
mxCycleTransitionState:=(miCycleState<>miCycleOldstate);
(*State text*)
sCycleStateText:=sCycleStateTextDef[miCycleState];
(*Timeout Watchdog for Statemachine*)
mxCycleTimeoutEnable:=NOT (miCycleState=0) AND NOT mxReset;

CycleTimeout(IN:=mxCycleTimeoutEnable, PT:=tCycleStateTimeouts[miCycleState] );
CycleTimeOutUpFlank(CLK:=CycleTimeout.Q );
miCycleOldstate:=miCycleState;

(*Set Errorbit when Raising edge of Timeout has been detected*)
IF CycleTimeOutUpFlank.Q THEN
	exCycleTimeOut:=TRUE; 			(* 1 Timeout for the whole programcycle *)
END_IF

(*Function to reset the Statemachine*)
IF mxResetCycleState THEN
	mxResetCycleState:= FALSE;
	mxInitialized:= FALSE;
	miCycleState:=0;
	miCycleOldstate:=miCycleState;
	mxCycleTransitionState:=FALSE;

	mxStartCycle:= FALSE;
	mxStopCycle:= FALSE;
	mxStopDirect:= FALSE;
	mxTakeoutIsMovingUp:= FALSE; 
	mxProductReadyAtTakeOut:= FALSE;
	mxSwitchVacuumOn:= FALSE;
	SgBottomIsIn := FALSE;
	SgBottomIsOut := FALSE;
	sgMoveIn := FALSE;
	sgMoveOut := FALSE;
	mxEmptyMachine := FALSE;
	
	
	mxProductOnTopMold:= FALSE;
	
	T_VCilinderMoveIn.IN :=FALSE;
	HorizontalAxis.M_Stop();
	
	//HydraulicCilinder.M_Stop();
END_IF

(*Definition State has Error*)
mxCycleHasError:=FALSE;

T_TakeOutTime(IN:=, PT:= MachParameters.VerticalCilinderTakeOutTime);
T_VCilinderMoveOut(IN:=, PT:= T#3S);
T_VCilinderMoveIn(IN:=, PT:=MachParameters.VerticalCilinderUpDelay);
T_VacuumBottomMoldClosed(IN:=, PT:=MachParameters.BottomMoldVacuumClosed);
RT_VacuumBottomMoldClosed(CLK:= MachParameters.ClosedVacEnabled AND SgMoldsAreClosed);
FT_SwitchVacuumOff(CLK:=mxSwitchVacuumOn);

IF RT_VacuumBottomMoldClosed.Q THEN
	T_VacuumBottomMoldClosed.IN:=TRUE;
	Vacuum.M_On();
END_IF

IF T_VacuumBottomMoldClosed.Q THEN
	T_VacuumBottomMoldClosed.IN:=FALSE;
	Vacuum.M_Off();
END_IF

(* Gantry picked up product from the Takeout unit *) 
RT_GantryPickedUpProduct(CLK:= mxGantryPickedUpProduct);

IF mxSwitchVacuumOn AND mxAutoMode THEN
	IF MachParameters.EnableVacuumSection[1] THEN VacuumTakeout[1].M_On(); END_IF
	IF MachParameters.EnableVacuumSection[2] THEN VacuumTakeout[2].M_On(); END_IF
	IF MachParameters.EnableVacuumSection[3] THEN VacuumTakeout[3].M_On(); END_IF
	IF MachParameters.EnableVacuumSection[4] THEN VacuumTakeout[4].M_On(); END_IF
END_IF 

IF FT_SwitchVacuumOff.Q AND mxAutoMode THEN
	IF MachParameters.EnableVacuumSection[1] THEN VacuumTakeout[1].M_Off(); END_IF
	IF MachParameters.EnableVacuumSection[2] THEN VacuumTakeout[2].M_Off(); END_IF
	IF MachParameters.EnableVacuumSection[3] THEN VacuumTakeout[3].M_Off(); END_IF
	IF MachParameters.EnableVacuumSection[4] THEN VacuumTakeout[4].M_Off(); END_IF
END_IF

IF (miCycleState >= 3 AND miCycleState <= 5) THEN	
		IF (ContinueWithA AND (ActualPositionTransfermold < (TransferPosA + MachParameters.StartVacAtTrPosOffset))) OR // At an ofset of transfermold pos
		 (ContinueWithB AND (ActualPositionTransfermold < (TransferPosB + MachParameters.StartVacAtTrPosOffset))) THEN	// Open the vacuum valve.
			Vacuum.M_On();
		END_IF
END_IF

(*Cycle State's*)
CASE miCycleState OF
{region "Description"}
	(*
		-Wait for move in signal from transfermold
		-Move in
		-Als product aan topmold, takeout unit up, vacuum aan, blow off topmold aan
		-wacht op transfer is down
		-vacuum aan
		-wacht op transfer is up
		-move Out
		-Set signal ready for takeout gantry
		-Set signal move topmold down
		-wait for Top mold is Up after drying
		-goto 1
	*)
{endregion}

	0:
	IF mxStartCycle THEN
			mxStartCycle:= FALSE;
			miCycleState:= 1;
	END_IF	

	1: // Wait for transfer/Drying ready to move in *)
		IF mxStopDirect THEN
			mxStopDirect:= FALSE;
			miCycleState:= 25;
		ELSIF mxStopCycle AND mxEmptyMachine THEN
			mxStopCycle:=False;
			mxEmptyMachine:= FALSE;
			miCycleState:= 0;
		ELSIF mxStopCycle THEN
			mxStopCycle:= FALSE;
			miStopState:= miCycleState;
			miCycleState:= 20;
		ELSIF SgMoveIn THEN
			SgMoveIn:= FALSE;
			SgBottomIsOut:= FALSE;
			
			miCycleState:= 2;
		END_IF

	2:	// Move IN
		IF mxStopDirect THEN
			mxStopDirect:= FALSE;
			miCycleState:= 25;
		ELSIF mxStopCycle THEN
			mxStopCycle:= FALSE;
			miStopState:= miCycleState;
			miCycleState:= 20;
		ELSIF HorizontalAxis.M_MoveAbsolute(MachParameters.AxisVelocityAuto, MachParameters.PositionInStop) AND HorizontalCilinder.M_In() THEN
			SgBottomIsIn:= TRUE;
			SgBottomIsOut := FALSE;
			MachParameters.KickOffCounter := MachParameters.KickOffCounter +1;
			
			miCycleState:=3;
		END_IF

	3:	// Move Take out vertical Up
		IF mxStopDirect THEN
			mxStopDirect:= FALSE;
			miCycleState:= 25;
		ELSIF mxStopCycle THEN
			mxStopCycle:= FALSE;
			miStopState:= miCycleState;
			miCycleState:= 20;
		ELSIF mxProductOnTopMold THEN									// check if there is a product
			T_VCilinderMoveIn.IN :=TRUE;
								
			IF (VerticalCilinder.M_In() OR T_VCilinderMoveIn.Q) THEN	// if there is a product, Get it with the cylinder.				
				mxTakeoutIsMovingUp:= TRUE;								// when cilinder is up signal topmold to start blowoff

				mxSwitchVacuumOn:= TRUE;
				T_VCilinderMoveIn.IN :=FALSE;
				
				miCycleState:= 4;
			END_IF
		ELSE 
			miCycleState:= 5;
		END_IF


	4:	// Move take out vertical down 	
		T_TakeOutTime.IN:= TRUE;
		mxTakeoutIsMovingUp:= FALSE;
		
		IF mxStopDirect THEN
			mxStopDirect:= FALSE;		
			miCycleState:= 25;
		ELSIF mxStopCycle THEN
			mxStopCycle:= FALSE;			
			miStopState:= miCycleState;
			miCycleState:= 20;
		ELSIF T_TakeOutTime.Q  THEN
			IF VerticalCilinder.M_Out() THEN
				T_TakeOutTime.IN:= FALSE;
				IF NOT mxEmptyMachine THEN
					miCycleState:= 5;
				ELSE
					miCycleState:= 6;
				END_IF
			END_IF
		END_IF		

	
	5: // Wait for transfer is down, vacuum on 
		IF mxStopDirect THEN
			mxStopDirect:= FALSE;
			miCycleState:= 25;
		ELSIF mxStopCycle THEN
			mxStopCycle:= FALSE;
			miStopState:= miCycleState;
			miCycleState:= 20;
		ELSIF sgMoveOut THEN	// When the closed wait time has elapsed and tranfer is up.
			sgMoveOut:= FALSE;
			miCycleState:= 6;
		END_IF
		
	6: // Move OUT, takeout horizontal out
		IF HorizontalAxis.ActPosition > (MachParameters.PositionOutStop - MachParameters.StopVacAtBmPosOffset) THEN
			Vacuum.M_Off();
		END_IF
	
		IF mxStopDirect THEN
			mxStopDirect:= FALSE;	
			miCycleState:= 25;
		ELSIF mxStopCycle THEN
			mxStopCycle:= FALSE;	
			miStopState:= miCycleState;
			miCycleState:= 20;
		ELSIF HorizontalAxis.M_MoveAbsolute(MachParameters.AxisVelocityAuto,MachParameters.PositionOutStop) AND HorizontalCilinder.M_Out() THEN
			SgBottomIsOut:= TRUE;
			SgBottomIsIn:= FALSE;
			mxSwitchVacuumOn:= FALSE;
			MachParameters.KickOffCounter := MachParameters.KickOffCounter +1;			
			IF mxProductOnTopMold THEN mxProductReadyAtTakeOut:= TRUE; END_IF
			miCycleState:= 7;
		END_IF

	7:	// Wait for product is picked up by gantry	
		IF mxStopDirect THEN
			mxStopDirect:= FALSE;
			miCycleState:= 25;
		ELSIF mxStopCycle THEN
			mxStopCycle:= FALSE;
			miStopState:= miCycleState;
			miCycleState:= 20;
		ELSIF (mxProductOnTopMold AND RT_GantryPickedUpProduct.Q) OR NOT mxProductOnTopMold THEN
			mxProductReadyAtTakeOut := FALSE; // -> stop signaling the gantry that there is a product ready to take
			mxProductOnTopMold:= FALSE;
			mxGantryPickedUpProduct:= FALSE;
		
			miCycleState:= 9;
		END_IF

	9: 	// Move Takeout IN 
		IF mxStopDirect THEN
			mxStopDirect:= FALSE;		
			miCycleState:= 25;
		ELSIF mxStopCycle THEN
			mxStopCycle:= FALSE;			
			miStopState:= miCycleState;
			miCycleState:= 20;
		ELSIF HorizontalCilinder.M_In() THEN
			miCycleState:= 1;
		END_IF

	20: // Stop Cycle, 
		IF mxStopDirect THEN
			mxStopDirect:= FALSE;		
			miCycleState:= 25;
		ELSIF TRUE THEN		
			miCycleState:= 21;
		END_IF

	21:	// Stop Cycle 
		IF mxStopDirect THEN
			mxStopDirect:= FALSE;
			miCycleState:= 25;
		ELSIF mxStartCycle THEN
			mxStartCycle:= FALSE;
			miCycleState:= miStopState;
		END_IF

	25: // Stop Direct 
		mxInitialized:= FALSE;

		mxStartCycle:= FALSE;
		mxStopCycle:= FALSE;
		mxStopDirect:= FALSE;
		
		mxTakeoutIsMovingUp:= FALSE; 
		mxSwitchVacuumOn:= FALSE;
		SgBottomIsIn := FALSE;
		SgBottomIsOut := FALSE;
		sgMoveIn := FALSE;
		sgMoveOut := FALSE;
		
		Vacuum.M_Off();
		
		miCycleState:= 0;
END_CASE

mxCycleBusy:= miCycleState<>0 AND NOT (miCycleState=21);
END_ACTION

ACTION Error:

FOR miVacSection:= 1 TO GVL.MaxNrOfVacSectTakeOutUnit DO
	T_VacSectionDelay[miVacSection](IN:= VacuumTakeout[miVacSection].mxIsOn, PT:= T#3S);
	SR_ErrorNoVacAtSection[miVacSection](SET1:= MachParameters.EnableVacuumSection[miVacSection] AND VacuumTakeout[miVacSection].mxIsOn AND 
	(T_VacSectionDelay[miVacSection].Q AND NOT VacuumSensor[miVacSection]), 
	RESET:= mxReset, Q1=> Errors.VacuumSection[miVacSection]);
END_FOR

(*************************************************************************************************)
mxErrorStopinPos:= HorizontalCilinder.mxErrorStopInPos OR VerticalCilinder.mxErrorStopInPos;
mxErrorInit:=HorizontalAxis.ErrorStop OR HorizontalCilinder.mxErrorInit  OR VerticalCilinder.mxErrorInit
			OR HeatingZone[1].mxErrorInit
			OR HeatingZone[2].mxErrorInit
			OR HeatingZone[3].mxErrorInit
			OR HeatingZone[4].mxErrorInit
			OR HeatingZone[5].mxErrorInit
			OR HEatingZone[6].mxErrorInit;
END_ACTION

ACTION Init:
(*StateChange (Transition)  Signalgeneration*)
mxInitTransitionState:=(miInitState<>miInitOldstate);
(*State text*)
sInitStateText:=sInitStateTextDef[miInitState];
(*Timeout Watchdog for Statemachine*)
mxInitTimeoutEnable:=NOT (miInitState=0)  AND NOT mxReset;

InitTimeout(IN:=mxInitTimeoutEnable  , PT:=tInitStateTimeouts[miInitState] );
InitTimeOutUpFlank(CLK:=InitTimeout.Q );
miInitOldstate:=miInitState;

(*Set Errorbit when Raising edge of Timeout has been detected*)
IF InitTimeOutUpFlank.Q THEN
	exInitTimeOut:=TRUE; 			(* 1 Timeout for the whole programcycle *)
END_IF

(*Function to reset the Statemachine*)
IF mxResetInitState THEN
	mxResetInitState:=FALSE;
	miInitState:=0;
	miInitOldstate:=miInitState;
	mxInitTransitionState:=FALSE;

	mxStartInit:= FALSE;
	mxStopInit:= FALSE;
	
END_IF

(*Definition State has Error*)
mxInitHasError:=FALSE;

(*Init State's*)
CASE miInitState OF
	0:
		IF mxStartInit THEN
			mxStartInit:= FALSE;
			mxInitialized:= FALSE;
			Vacuum.M_Off();
			mxSwitchVacuumOn:= FALSE;
			
			miInitState:= 1;
		END_IF

	(* Vertical cilinder Down *)
	1:
		IF mxStopInit THEN
			mxStopInit:= FALSE;
			
			miInitState:= 10;
		ELSIF VerticalCilinder.M_Out() THEN	(*BaTeu, changed M_in to M_out (In = Up / out = down) *)
			
			miInitState:= 2;
		END_IF
	
	(* Move OUT *)
	2:
		IF mxStopInit THEN
			mxStopInit:= FALSE;
			
			miInitState:= 10;
		ELSIF HorizontalAxis.M_MoveAbsolute(MAchparameters.AxisVelocityInit, MachParameters.PositionOutStop) THEN

			miInitState:= 3;
		END_IF

	(* Horizontal cilinder Out *)
	3:
		IF mxStopInit THEN
			mxStopInit:= FALSE;
			
			miInitState:= 10;
		ELSIF HorizontalCilinder.M_Out() THEN

			mxInitialized:= TRUE;
			miInitState :=0;
		END_IF	

	(* Stop Init *)
	10:
		HorizontalAxis.M_Stop();
		mxStartInit:= FALSE;
		mxStopInit:= FALSE;
		mxInitialized:= FALSE;
		
		miInitState:= 0;
			
END_CASE

mxInitBusy:= miInitState<>0;
END_ACTION

METHOD M_EmptyMachine

IF mxCycleBusy THEN
	mxEmptyMachine:= TRUE;	
END_IF
END_METHOD

METHOD M_StartCycle

IF NOT mxCycleBusy THEN
	mxStopCycle := FALSE;
	mxStartCycle:= TRUE;	
END_IF
END_METHOD

METHOD M_StartInit

IF NOT mxInitBusy THEN 
	mxStartInit:= TRUE; 
END_IF
END_METHOD

METHOD M_StopCycle

IF mxCycleBusy THEN 
	mxStopCycle:= TRUE; 
END_IF
END_METHOD

METHOD M_StopDirect

IF mxCycleBusy THEN
	mxStopDirect:= TRUE;	
END_IF
END_METHOD

METHOD M_StopInit

IF mxInitBusy THEN 
	mxStopInit:= TRUE; 
END_IF
END_METHOD

ACTION Objects:
HorizontalAxis(
	mxEnable:= NOT mxEmergency OR NOT mxDoorsOpened, 
	mxInhibit:= RHSR_Blocked, //20190124 (was hard FALSE).
	mxAutoMode:= mxAutoMode, 
	mxReset:= mxReset, 
	mxFirstCycle:= mxFirstCycle, 
	mxEmergency:= mxEmergency, 
	mxSimulation:= , 
	mxResetCycle:= , 
	mxDisable_Positive:= FALSE,
	mxDisable_Negative:= FALSE,
	mxBlockHMI:= , 
	mrOverride:=100.0 , 
	mrVelocityManual:= MachParameters.AxisVelocityManual,  
	mrHomePos:= MachParameters.AxisPositionHome, 
	SysParameters:= SysParameters.BottomMoldAxis,
	mxAxisIsMoving=> mrAxisIsMoving, 
	Errors=> Errors.HorizontalAxis, 
	ActPosition=>mrAxisActPos );
	
Vacuum(
	mxReset:= mxReset, 
	mxEmergency:= mxEmergency OR mxDoorsOpened, 
	mxAutoMode:= mxAutoMode);

VacuumTakeout[1](
	mxReset:=mxReset , 
	mxEmergency:= mxEmergency OR mxDoorsOpened, 
	mxAutoMode:=mxAutoMode , 
	mxIsOn=>);

VacuumTakeout[2](
	mxReset:=mxReset , 
	mxEmergency:= mxEmergency OR mxDoorsOpened, 
	mxAutoMode:=mxAutoMode , 
	mxIsOn=>);
	
VacuumTakeout[3](
	mxReset:=mxReset , 
	mxEmergency:= mxEmergency OR mxDoorsOpened, 
	mxAutoMode:=mxAutoMode , 
	mxIsOn=>);
	
VacuumTakeout[4](
	mxReset:=mxReset , 
	mxEmergency:= mxEmergency OR mxDoorsOpened, 
	mxAutoMode:=mxAutoMode , 
	mxIsOn=>);
	
VacuumTakeout[5](
	mxReset:=mxReset , 
	mxEmergency:= mxEmergency OR mxDoorsOpened, 
	mxAutoMode:=mxAutoMode , 
	mxIsOn=>);	
	
VacuumTakeout[6](
	mxReset:=mxReset , 
	mxEmergency:= mxEmergency OR mxDoorsOpened, 
	mxAutoMode:=mxAutoMode , 
	mxIsOn=>);
		
(* Take out Unit *)
HorizontalCilinder(
	mxReset:= mxReset, 
	mxEmergency:=  mxEmergency OR mxDoorsOpened, 
	mxAutoMode:= mxAutoMode, 
	MachParameters:= MachParameters.HorizontalCilinder, 
	mxIsVertical:=FALSE,
	mxIsIn=> mxHorCilIsIn, 
	mxIsOut=> mxHorCilIsOut, 
	Errors=> Errors.HorizontalCilinder);
	
VerticalCilinder(
	mxReset:= mxReset, 
	mxEmergency:=  mxEmergency OR mxDoorsOpened, 
	mxAutoMode:= mxAutoMode, 
	MachParameters:= MachParameters.VerticalCilinder, 
	mxIsVertical:=TRUE,
	mxIsIn=> mxVertCilIsIn, 
	mxIsOut=> mxVertCilIsOut, 
	Errors=> Errors.VerticalCilinder);

HeatingZone[1](
	mxReset:= mxReset,
	mxEmergency:=mxEmergency,
	mxDoorsOpened:=mxDoorsOpened,
	mxEnableHeating:=mxEnableHeating,
	MachParameters:=MachParameters.HeatingZone[1],
	Errors=> Errors.HeatingZone[1]);

HeatingZone[2](
	mxReset:= mxReset,
	mxEmergency:=mxEmergency,
	mxDoorsOpened:=mxDoorsOpened,
	mxEnableHeating:=mxEnableHeating,
	MachParameters:=MachParameters.HeatingZone[2],
	Errors=> Errors.HeatingZone[2]);

HeatingZone[3](
	mxReset:= mxReset,
	mxEmergency:=mxEmergency,
	mxDoorsOpened:=mxDoorsOpened,
	mxEnableHeating:=mxEnableHeating,
	MachParameters:=MachParameters.HeatingZone[3],
	Errors=> Errors.HeatingZone[3]);

HeatingZone[4](
	mxReset:= mxReset,
	mxEmergency:=mxEmergency,
	mxDoorsOpened:=mxDoorsOpened,
	mxEnableHeating:=mxEnableHeating,
	MachParameters:=MachParameters.HeatingZone[4],
	Errors=> Errors.HeatingZone[4]);

HeatingZone[5](
	mxReset:= mxReset,
	mxEmergency:=mxEmergency,
	mxDoorsOpened:=mxDoorsOpened,
	mxEnableHeating:=mxEnableHeating,
	MachParameters:=MachParameters.HeatingZone[5],
	Errors=> Errors.HeatingZone[5]);

HeatingZone[6](
	mxReset:= mxReset,
	mxEmergency:=mxEmergency,
	mxDoorsOpened:=mxDoorsOpened,
	mxEnableHeating:=mxEnableHeating,
	MachParameters:=MachParameters.HeatingZone[6],
	Errors=> Errors.HeatingZone[6]);
END_ACTION

END_FUNCTION_BLOCK

// ---- POUs/Standard/Valves/FB_BiValve2Fdbck.TcPOU
FUNCTION_BLOCK FB_BiValve2Fdbck
VAR_INPUT
	mxReset						: BOOL;	(*Reset Error*)
	mxEmergency					: BOOL;
	mxAutoMode					: BOOL; (* TRUE = Automode *)
	mxCheckCilinder				: BOOL:= TRUE;
	mxIsVertical				: BOOL;
END_VAR
VAR_IN_OUT
	MachParameters					: ST_CilinderParameters;
END_VAR
VAR_OUTPUT
	mxIsIn						: BOOL;
	mxIsOut						: BOOL;
	mxIsOpen					: BOOL;
	mxIsClosed					: BOOL;
	Errors						: ST_CilinderErrors;
	
	mxErrorInit: BOOL;
	mxErrorStopInPos: BOOL;

END_VAR
VAR
	Check						: FB_CheckCilinder;
	
	QxIn	 					AT %Q*: BOOL;
	QxOut						AT %Q*: BOOL;
	IxIsIn						AT %I*: BOOL;
	IxIsOut						AT %I*: BOOL;

	mxHMI_In					: BOOL;
	mxHMI_Out					: BOOL;
	mxHMI_Open					: BOOL;
	mxHMI_Close					: BOOL;
	RT_HMI_In					: R_TRIG;
	RT_HMI_Out					: R_TRIG;
END_VAR

Error();

RT_HMI_In(CLK:= NOT mxAutoMode AND (mxHMI_In OR mxHMI_Open));
RT_HMI_Out(CLK:= NOT mxAutoMode AND (mxHMI_Out OR mxHMI_Close));

(* Manual *)
IF RT_HMI_In.Q THEN M_In(); END_IF
IF RT_HMI_Out.Q THEN M_Out(); END_IF

(* Reset Outputs *)

//IF IxIsIn THEN QxIn:= FALSE; END_IF
//IF IxIsOut THEN QxOut:= FALSE; END_IF

(* Status *)
mxIsIn:= mxIsOpen:= IxIsIn;
mxIsOut:= mxIsClosed:= IxIsOut;

ACTION Error:

IF NOT mxIsVertical THEN
	
	Check(
		MoveCilOut:= qxOut,
		MoveCilin:= qxIn,
		CheckCilinder:= mxCheckCilinder,
		SensorOut:=  mxIsOut OR mxIsClosed, // mx closed and open omgedraaid (20180528 -> Bateu*)
		SensorIn:= mxIsIn OR mxIsOpen,
		TimMax:= MachParameters.T_GuardTimeError,
		mxReset:= mxReset,
		ErrorCilinder=> Errors.Cilinder,
		ErrorCilinderOut=> ,
		ErrorCilinderIn=> ,
		ErrorEndNotReached=> ,
		ErrorSensorSwitched=> ,
		Time_Cil_Out=> ,
		Time_Cil_In=> );

(* Too slow errors, only messages *)

	Errors.CilinderSlow_IN	:=	mxCheckCilinder AND (Check.Time_Cil_In > MachParameters.T_GuardTimeWarning_IN);
	Errors.CilinderSlow_OUT	:=	mxCheckCilinder AND (Check.Time_Cil_Out > MachParameters.T_GuardTimeWarning_OUT);
END_IF

(**********************************************************************************************************)
mxErrorStopinPos:= FALSE;
mxErrorInit:= Errors.Cilinder;
END_ACTION

METHOD PUBLIC M_Close: BOOL
VAR_INPUT
END_VAR

IF NOT IxIsOut THEN QxOut:= TRUE; END_IF
QxIn:= FALSE;

(* Return value *)
M_Close:= IxIsOut;
END_METHOD

METHOD PUBLIC M_In : BOOL
VAR_INPUT
END_VAR

IF NOT IxIsIn THEN QxIn:= TRUE; END_IF
//QxIn:= TRUE;
QxOut:= FALSE;

(* Return value *)
M_In:= IxIsIn;
END_METHOD

METHOD PUBLIC M_In_Pressure : BOOL
VAR_INPUT
END_VAR
QxIn:= TRUE;
QxOut:= FALSE;

(* Return value *)
M_In_Pressure:= IxIsIn;
END_METHOD

METHOD PUBLIC M_Open : BOOL
VAR_INPUT
END_VAR

IF NOT IxIsIn THEN QxIn:= TRUE; END_IF
QxOut:= FALSE;

(* Return value *)
M_Open:= IxIsIn;
END_METHOD

METHOD PUBLIC M_Out: BOOL
VAR_INPUT
END_VAR

IF NOT IxIsOut THEN QxOut:= TRUE; END_IF
//qxOut:=TRUE;
QxIn:= FALSE;

(* Return value *)
M_Out:= IxIsOut;
END_METHOD

END_FUNCTION_BLOCK

// ---- POUs/Standard/Valves/FB_CheckCilinder.TcPOU
FUNCTION_BLOCK FB_CheckCilinder

VAR_INPUT
	mxReset:BOOL;					(* Reset error *)	
	MoveCilOut:BOOL; 				(* Set output cilinder out *)
	MoveCilin:BOOL; 				(* Set output cilinder in *)
	CheckCilinder: BOOL;			(* Cilinder is enabled *)
	SensorOut:BOOL; 				(* Sensor cilinder out *)
	SensorIn:BOOL; 					(* Sensor cilinder in *)
	TimMax:TIME;					(* Maximum moving time *)
END_VAR

VAR_OUTPUT
	ErrorCilinder:BOOL;				(* Error cilinder not in position *)
	ErrorCilinderOut: BOOL;			(* Error cilinder not in position out *)
	ErrorCilinderIn: BOOL;			(* Error cilinder not in position in *)
	ErrorEndNotReached:BOOL;		(* Error cilinder was not in endposition at new comand *)
	ErrorSensorSwitched:BOOL;		(* Error sensor switched off after in position *)
	Time_Cil_Out:TIME;			(* Duration cilinder moving *)
	Time_Cil_In:TIME;				(* Duration cilinder moving *)

END_VAR

VAR
	CilinderOut:BOOL;				(* Helpbit last positioncommand *)
	CilinderIn:BOOL;				(* Helpbit last positioncommand *)
	
	PositionOut:BOOL;				(* Last position detected is out *)
	PositionIn:BOOL;				(* Last position detected is in *)
	fbiTimMaxOut:TON;				(* Maximum movingtime *)
	fbiTimMaxIn:TON;				(* Maximum movingtime *)
	fbiTim_Check_Sens: TON;		(* Check both sensors on *)
	R_TrigCilOut:R_TRIG;			(* Puls command cilinder out *)
	R_TrigCilin:R_TRIG;				(* Puls command cilinder in *)
	R_TrigSensOut:R_TRIG;			(* Puls cilinder comes in position out *)
	R_TrigSensIn:R_TRIG;			(* Puls cilinder comes in position in *)
	F_TrigSensOut:F_TRIG;			(* Puls cilinder was in position out *)
	F_TrigSensIn:F_TRIG;			(* Puls cilinder was in position in *)

	LastPosOut: BOOL;		(*Last command before this new one*)
	fbiTime_Out: TOF;		(* Duration cilinder moving out *)
	fbiTime_In: TOF;			(* Duration cilinder moving in *)
	T_SensorOut			: TOF;
	T_SensorIn			: TOF;

	LastTime_Cil_Out:TIME;			(* Duration cilinder moving, on HMI *)
	LastTime_Cil_In:TIME;				(* Duration cilinder moving, on HMI *)
END_VAR

(* Store last position command *)
IF MoveCilOut THEN CilinderOut:=TRUE; CilinderIn:=FALSE;	END_IF
IF MoveCilin THEN CilinderIn:=TRUE;	 CilinderOut:=FALSE; END_IF

(* Puls command cilinder in/out *)
R_TrigCilOut(CLK:=CilinderOut);
R_TrigCilin(CLK:=CilinderIn);

(* Puls sensor in/out *)
T_SensorIn(IN:= SensorIn, PT:= T#500ms);
T_SensorOut(IN:= SensorOut, PT:=T#500ms);
R_TrigSensOut(CLK:=SensorOut);
F_TrigSensOut(CLK:=SensorOut);
R_TrigSensIn(CLK:=SensorIn);
F_TrigSensIn(CLK:=SensorIn);

(* Check if sensor switched off after in position *)
IF CheckCilinder THEN
	IF (CilinderOut AND F_TrigSensOut.Q) OR (CilinderIn AND F_TrigSensIn.Q)  THEN
		ErrorCilinder:=TRUE;
		ErrorSensorSwitched:=TRUE;
	END_IF
END_IF

(******************************************************************************
Cilinder in or out: Check movingtime & other sensor is off
******************************************************************************)
fbiTimMaxOut(IN:=CilinderOut AND CheckCilinder,PT:=TimMax);
IF fbiTimMaxOut.Q AND ( SensorIn OR NOT SensorOut) THEN
	ErrorCilinder:=TRUE;
	ErrorCilinderOut:=TRUE;
END_IF

fbiTimMaxIn(IN:=CilinderIn AND CheckCilinder,PT:=TimMax);
IF fbiTimMaxIn.Q AND ( SensorOut OR NOT SensorIn) THEN
	ErrorCilinder:=TRUE;
	ErrorCilinderIn:=TRUE;
END_IF


(******************************************************************************
Check if both sensors on
******************************************************************************)
fbiTim_Check_Sens(IN:=SensorOut AND SensorIn AND CheckCilinder, PT:=TimMax);
IF fbiTim_Check_Sens.Q THEN
	ErrorCilinder:=TRUE;
	ErrorCilinderOut:=TRUE;
	ErrorCilinderIn:=TRUE;
END_IF

(******************************************************************************
Check if sensors was on before switch-over to other side
******************************************************************************)
IF R_TrigCilOut.Q AND NOT LastPosOut AND NOT SensorIn THEN
	ErrorEndNotReached:=TRUE;
END_IF
IF R_TrigCilin.Q AND LastPosOut AND NOT SensorOut THEN
	ErrorEndNotReached:=TRUE;
END_IF
IF R_TrigCilOut.Q THEN LastPosOut:=TRUE; END_IF
IF R_TrigCilin.Q THEN LastPosOut:=FALSE; END_IF


(******************************************************************************
Reset Errors
******************************************************************************)
IF mxReset THEN
	ErrorCilinder:=FALSE;
	ErrorCilinderOut:=FALSE;
	ErrorCilinderIn:=FALSE;
	ErrorEndNotReached:=FALSE;
	ErrorSensorSwitched:=FALSE;
END_IF


(******************************************************************************
Timers for display actual movingtime
******************************************************************************)
(* preset timer on startcommand *)
fbiTime_Out(IN:=R_TrigCilOut.Q,PT:=t#60s);
fbiTime_In(IN:=R_TrigCilin.Q,PT:=t#60s);
(* Display actual movingtime *)
IF R_TrigSensOut.Q THEN
	Time_Cil_Out:=fbiTime_Out.ET;
	LastTime_Cil_Out:=fbiTime_Out.ET;
ELSIF mxReset THEN
	Time_Cil_Out:= T#0ms;
END_IF
IF R_TrigSensIn.Q THEN
	Time_Cil_In:=fbiTime_In.ET;
	LastTime_Cil_In:=fbiTime_In.ET;
ELSIF mxReset THEN
	Time_Cil_In:= T#0ms;
END_IF

END_FUNCTION_BLOCK

// ---- POUs/Standard/NC_Axis/FB_NcAxis.TcPOU
FUNCTION_BLOCK FB_NcAxis
VAR CONSTANT

	sPosBiasStateTextDef: ARRAY[0..2] OF STRING:=	['State 0: Wait for Start',
										'State 1: Read Pos Bias, calculate new Pos Bias',
										'State 2: Write Pos Bias'];

	tPosBiasStateTimeouts: ARRAY[0..2] OF TIME:=  [T#10S, T#10S, T#10S];
	
END_VAR
VAR_INPUT
	mxEnable						: BOOL;
	mxInhibit						: BOOL :=TRUE;
	mxAutoMode						: BOOL;
	mxReset							: BOOL;
	mxFirstCycle					: BOOL;
	mxEmergency						: BOOL;
	mxSimulation					: BOOL;
	mxResetCycle					: BOOL;
	mxDisable_Positive				: BOOL; 
	mxDisable_Negative				: BOOL;
	mxBlockHMI						: BOOL:= FALSE;
	mrOverride						: LREAL;
	mrVelocityManual				: LREAL;
	mxResetPosBiasState				: BOOL;
	mxZeroCommand					: BOOL;
	mrHomePos						: LREAL;
END_VAR
VAR_IN_OUT
	SysParameters					: ST_NcAxis_SysPar;
END_VAR
VAR_OUTPUT
	mxCycleBusy						: BOOL;
	mxRunning						: BOOL;
	mxAxisIsMoving					: BOOL;
	///Errors
	Errors							: st_NcAxis_Errors;
	Error							: BOOL;
	ErrorStop						: BOOL;

	axStatus						:ST_AxisStatus;
	ActPosition						:LREAL;
	ActVelocity						:LREAL;

	axAxis							: AXIS_REF;

	mxPosBiasBusy					: BOOL;
	mxPosBiasHasError				: BOOL;
	SignalLightStatus					: BOOL;(* Needed in the HMI, for changing the color of the signal light *)	
END_VAR
VAR
	HmiStatus: UINT;
	HmiControl: UINT;
	HMI_ReadEncoder:BOOL;
	HMI_ReadmInc:LREAL;
	HMI_WriteEncoder:BOOL;
	HMI_WritemInc: LREAL;
	
	HMI_Forward				: BOOL;
	HMI_Backward			: BOOL;
	mxActivateAuto:BOOL;
	mxActivateManual:BOOL;
	mxActivated:BOOL;
	
	MCPower							: MC_Power;
	MCReset							: MC_Reset;
	MCJog							: MC_Jog;
	MCStop							: MC_Stop;
	MCHome							: MC_Home;
	MCMoveAbsolute					: ARRAY[0..1] OF MC_MoveAbsolute;
	mxMoveAbsNr						: INT;
	MCMoveVelocity					: ARRAY[0..1] OF MC_MoveVelocity;
	mxMoveVelocityNr				: INT;	
	MCReadParameter					: MC_ReadParameter;
	MCReadAxisError					: MC_ReadAxisError;
	MCWriteParameter				: MC_WriteParameter; 
 	MCSetPosition					: MC_SetPosition;
	MCReadStatus					: MC_ReadStatus;
	mcResetDrive					: FB_SoEReset_ByDriveRef;
	iDriveRef						AT %I* :ST_PLCDriveRef;
	
(*Drive parameters*)	
	mcBlendingMode					: MC_BufferMode;

	miState							: INT	:=0;
	miStopState						: INT	:=0;
	miOldstate						: INT	:=0;
	mxTransitionState				: BOOL	:= FALSE;
	sStateText						: STRING;	
	
 	exPosBiasTimeOut				: BOOL;		(* Timeout for the whole programcycle *)
	miPosBiasState					: INT	:=0;
	miPosBiasOldstate				: INT	:=0;
	mxPosBiasTransitionState		: BOOL	:= FALSE;
	sPosBiasStateText				: STRING;
	PosBiasTimeout					: TON;

(* Vars *)
	mxPosBiasTimeoutEnable			: BOOL;
	PosBiasTime						: REAL;

	mrStoredAxisPosition			: LREAL;
	mxPositionError					: BOOL;

	AdsReadPosBias					: ADSREAD;
	AdsWritePosBias					: ADSWRITE;

	PositionBiasRead 				: LREAL;
	
	(* Errors *)
	SR_DrivePower					: SR;
	SR_DriveJog						: SR;
	SR_DriveStatus					: SR;
	SR_DriveStop					: SR;
	SR_DriveReset					: SR;
	SR_Home							: SR;
	SR_Restart						: SR;
	SR_MotorError					: SR;
	SR_DriveAbsError				: SR;
	SR_DriveVelocity				: SR;
	SR_WriteParameter				: SR;
	SR_ReadParameter				: SR;
	SR_LagError						: SR;

	
	mxCycleHasError					: BOOL;
	
(*Timers*)
	T_Power_On						: TON;
	T_Power_Off						: TOF;
	CycleTimeout					: TON;

(*Raising Edge detections*)
	RT_AutoManual					: R_TRIG;
	FT_AutoManual					: F_TRIG;
	RT_AutoManualHMI				: R_TRIG;
	CycleTimeOutUpFlank				: R_TRIG;
	PosBiasTimeOutUpFlank			: R_TRIG;

(* Vars *)
	mxCycleTimeoutEnable			: BOOL;
	CycleTime						: REAL;
	SR_CycleTimeOut					: SR;	
	mrPosition: LREAL;
	mrCheckPosition: LREAL;
	mxMoveForw: BOOL;
	mxSimulationDO	:INT:=0;	(*0= direct onposition, 1=seconds OnPosition, 2=not on position first and second*)
	ErrorIDMoveAbs1: UDINT;
	ErrorIDMoveAbs0: UDINT;

	T_Delay: TON;
	T_StandstillDelay: TON;
	miReadErrorID: DWORD;
	miReadAxisErrorID: DWORD;
END_VAR

Alarms();
WritePosBias();
HMI();
DriveActions();

ACTION Alarms:
SR_DrivePower(SET1:=MCPower.Error , RESET:=mxReset , Q1=> errors.exDrivePower);
SR_DriveJog(SET1:= MCJog.Error, RESET:=mxReset , Q1=> errors.exDriveJog);
SR_DriveStatus(SET1:= axAxis.Status.Error, RESET:=mxReset , Q1=> errors.exDriveStatus);
SR_DriveReset(SET1:= MCReset.Error, RESET:= mxReset, Q1=>errors.exDriveReset );
SR_DriveAbsError(SET1:=MCMoveAbsolute[0].Error OR MCMoveAbsolute[1].Error, RESET:= mxReset, Q1=>errors.exDriveAbsoluut );
SR_DriveStop(SET1:= MCStop.Error, RESET:= mxReset, Q1=>errors.exDriveStop );
SR_WriteParameter(SET1:= MCWriteParameter.Error, RESET:= mxReset, Q1=>errors.exWriteParameter );
SR_ReadParameter(SET1:= MCReadParameter.Error, RESET:= mxReset, Q1=>errors.exReadParameter );
SR_Home(SET1:= MCHome.Error, RESET:= mxReset, Q1=>errors.exHome );
SR_DriveVelocity(SET1:= MCMoveVelocity[0].Error OR MCMoveVelocity[0].Error, RESET:= mxReset, Q1=> Errors.exDriveVelocity);
SR_LagError(SET1:=(MCMoveAbsolute[0].ErrorID = 17744 AND MCMoveAbsolute[0].Error) OR 
						 (MCMoveAbsolute[1].ErrorID = 17744 AND MCMoveAbsolute[1].Error) OR
						 (MCJog.ErrorID = 17744 AND MCJog.Error) OR 
						 (MCMoveVelocity[0].ErrorID = 17744 AND MCMoveVelocity[0].Error) OR 
						 (MCMoveVelocity[1].ErrorID = 17744 AND MCMoveVelocity[1].Error) OR
						 axStatus.ErrorID = 17744
						 , RESET:= mxReset, Q1=>errors.exLagError );

ErrorStop:= errors.exLagError OR errors.exWriteParameter OR errors.exReadParameter OR 
	errors.exDriveStop OR errors.exDrivePower OR errors.exDriveJog  OR  errors.exDriveStatus OR 
	errors.exDriveReset OR Errors.exDriveAbsoluut OR Errors.exDriveVelocity OR errors.exHome;
END_ACTION

ACTION DriveActions:
(*read axis status*)
axAxis.ReadStatus();
axStatus:= axAxis.Status;
ActPosition:=axAxis.NcToPlc.ActPos;
ActVelocity:=axAxis.NcToPlc.ActVelo;
mxAxisIsMoving:= axAxis.Status.Moving;

	(*Power Axis*)
T_Power_On(IN:=(NOT mxInhibit), PT:= T#10MS);
T_Power_Off(IN:=T_Power_On.Q , PT:=T#5S , Q=> , ET=> );
(*power axis*)	
MCPower(
	Axis:= axAxis, 
	Enable:=NOT mxEmergency AND (T_Power_On.Q OR T_Power_Off.Q),  
	Enable_Positive:= NOT mxDisable_Positive , 
	Enable_Negative:= NOT mxDisable_Negative , 
	Override:=, 
	BufferMode:= , 
	Options:= , 
	Status=> , 
	Busy=> , 
	Active=> , 
	Error=> , 
	ErrorID=> );
	 
(*Drive run action manual*)
MCJog(
	Axis:= axAxis, 
	JogForward:= ,
	JogBackwards:= ,
	Mode:=MC_JOGMODE_CONTINOUS , 
	Position:= , 
	Velocity:= mrVelocityManual, 
	Acceleration:= , 
	Deceleration:= , 
	Jerk:= , 
	Done=> , 
	Busy=> , 
	Active=> , 
	CommandAborted=> , 
	Error=> , 
	ErrorID=> );
	MCJog.JogForward:=FALSE; 	
	MCJog.JogBackwards:=FALSE;

(*Drive Reset*)
MCReset(
	Axis:=axAxis , 
	Execute:=(mxReset AND (axAxis.Status.Error OR Error)), 
	Done=> , 
	Busy=> , 
	Error=> , 
	ErrorID=> );

	(*Reset*)
//DriveAxis.mcReset(Execute:= mxReset AND DriveAxis.mcStatus.Error, Axis:= axAxis);

(* Reset Drive Error *)
mcResetDrive.stDriveRef.sNetId:= F_CreateAmsNetId(iDriveRef.aNetId);
mcResetDrive.stDriveRef.nSlaveAddr:= iDriveRef.nSlaveAddr;
mcResetDrive.stDriveRef.nDriveNo:= iDriveRef.nDriveNo;


mcResetDrive(
	bExecute:= mxReset AND axAxis.Status.DriveDeviceError,
	tTimeout:= t#10s);
	
(*Move absolute fb 1*) 
	MCMoveAbsolute[0](
			Axis:= axAxis, 
			Execute:=, 
			Position:= , 
			Velocity:= , 
			Acceleration:= , 
			Deceleration:= , 
			Jerk:= , 
			BufferMode:= , 
			Options:= , 
			Done=> , 
			Busy=> , 
			Active=> , 
			CommandAborted=> , 
			Error=> , 
			ErrorID=> );
MCMoveAbsolute[0].Execute:=FALSE;
IF MCMoveAbsolute[0].ErrorID > 0 THEN ErrorIDMoveAbs0:=MCMoveAbsolute[0].ErrorID; END_IF;
(*Move absolute fb 2*)
	MCMoveAbsolute[1](
			Axis:= axAxis, 
			Execute:=, 
			Position:= , 
			Velocity:= , 
			Acceleration:= , 
			Deceleration:= , 
			Jerk:= , 
			BufferMode:=, 
			Options:= , 
			Done=> , 
			Busy=> , 
			Active=> , 
			CommandAborted=> , 
			Error=> , 
			ErrorID=>ErrorIDMoveAbs1 );
MCMoveAbsolute[1].Execute:=FALSE;
IF MCMoveAbsolute[1].ErrorID > 0 THEN ErrorIDMoveAbs0:=MCMoveAbsolute[1].ErrorID; END_IF;
(*Move velocity fb 1*)
MCMoveVelocity[0](
	Axis:=axAxis , 
	Execute:= , 
	Velocity:= , 
	Acceleration:= , 
	Deceleration:= , 
	Jerk:= , 
	Direction:= , 
	BufferMode:= , 
	Options:= , 
	InVelocity=> , 
	Busy=> , 
	Active=> , 
	CommandAborted=> , 
	Error=> , 
	ErrorID=> );
			
MCMoveVelocity[0].Execute:=FALSE;		
 (*Move velocity fb 2*)
MCMoveVelocity[1](
	Axis:=axAxis , 
	Execute:= , 
	Velocity:= , 
	Acceleration:= , 
	Deceleration:= , 
	Jerk:= , 
	Direction:= , 
	BufferMode:= , 
	Options:= , 
	InVelocity=> , 
	Busy=> , 
	Active=> , 
	CommandAborted=> , 
	Error=> , 
	ErrorID=> );
			
MCMoveVelocity[1].Execute:=FALSE;		

MCStop(
	Axis:=axAxis , 
	Execute:= , 
	Deceleration:= , 
	Jerk:= , 
	Options:= , 
	Done=> , 
	Busy=> , 
	Active=> , 
	CommandAborted=> , 
	Error=> , 
	ErrorID=> );
MCStop.Execute:=FALSE;

(*Homing*)
MCHome(
	Axis:=axAxis , 
	Execute:= , 
	Position:=  , 
	HomingMode:=  , 
	BufferMode:= , 
	Options:= , 
	bCalibrationCam:= , 
	Done=> , 
	Busy=> , 
	Active=> , 
	CommandAborted=> , 
	Error=> , 
	ErrorID=> );
MCHome.Execute:=FALSE;
	
(*Read a parameter*)
MCReadParameter(
	Axis:=axAxis , 
	Enable:= , 
	ParameterNumber:= , 
	ReadMode:=E_ReadMode.READMODE_CYCLIC , 
	Valid=> , 
	Busy=> , 
	Error=> , 
	ErrorID=> , 
	Value=> );
MCReadParameter.Enable:=FALSE;

(*Write a parameter*)	
MCWriteParameter(
	Axis:= axAxis, 
	Execute:= , 
	ParameterNumber:= , 
	Value:= , 
	Done=> , 
	Busy=> , 
	Error=> , 
	ErrorID=> );
MCWriteParameter.Execute:=FALSE;

MCSetPosition(
	Axis:= axAxis, 
	Execute:= , 
	Position:= , 
	Mode:=FALSE , 
	Options:= , 
	Done=> , 
	Busy=> , 
	Error=> , 
	ErrorID=> );
	MCSetPosition.Execute:=FALSE;	

MCReadAxisError(
	Axis:=axAxis , 
	Enable:=TRUE , 
	Valid=> , 
	Busy=> , 
	Error=> , 
	ErrorID=> miReadErrorID, 
	AxisErrorID=>miReadAxisErrorID );
	(*
MCReadStatus(
	Axis:= axAxis, 
	Enable:= , 
	Valid=> , 
	Busy=> , 
	Error=> , 
	ErrorID=> , 
	ErrorStop=> , 
	Disabled=> , 
	Stopping=> , 
	StandStill=> , 
	DiscreteMotion=> , 
	ContinuousMotion=> , 
	SynchronizedMotion=> , 
	Homing=> , 
	ConstantVelocity=> , 
	Accelerating=> , 
	Decelerating=> , 
	Status=> );*)
END_ACTION

ACTION HMI:
(*Read ax encoder parameter minc*)
IF HMI_ReadEncoder THEN
	HMI_ReadmInc :=	M_ReadParameter(MC_AxisParameter.AxisEncoderScalingFactor);
END_IF
(*Write ax encoder parameter*)
IF HMI_WriteEncoder THEN
	M_WriteParameter(miParameterNr:=MC_AxisParameter.AxisEncoderScalingFactor , miValue:= HMI_WritemInc );
END_IF

IF mxAutoMode THEN
	MCPower.Override:=mrOverride;
ELSE
	MCPower.Override:=mrOverride(*parameters.VelocityManual*);		
END_IF;

RT_AutoManual(CLK:= mxAutoMode);
FT_AutoManual(CLK:= mxAutoMode);

(*Set output*)
mxActivateAuto:= (mxEnable AND mxAutomode);
mxActivateManual := (mxEnable AND NOT mxAutoMode);

IF HMI_Forward AND axAxis.Status.Operational AND NOT SR_Restart.Q1 AND T_Power_On.Q AND NOT mxAutomode THEN
	MCJog.JogForward := TRUE ;
	MCJog.Velocity:= mrVelocityManual;
END_IF
IF HMI_Backward AND axAxis.Status.Operational AND NOT SR_Restart.Q1 AND T_Power_On.Q AND NOT mxAutoMode THEN
	MCJog.JogBackwards :=TRUE;
	MCJog.Velocity:= mrVelocityManual;
END_IF
END_ACTION

METHOD M_Home : BOOL;
VAR_INPUT
	mrHomePosition		: LREAL;
	MCMode				: MC_HomingMode;
END_VAR
McHome.Position:= mrHomePosition;
McHome.HomingMode:= MCMode;

McHome.Execute:= TRUE;


(* Return Value *)
M_Home:=MCHome.Done;
END_METHOD

METHOD M_MoveAbsolute : BOOL
VAR_INPUT
	Velocity				:LREAL;			
	Position				:LREAL;
END_VAR
(*compare for different setpoints, if so change fb mcMoveAbsolute*)
IF 	(MCMoveAbsolute[mxMoveAbsNr].Position <> Position) OR 
	(MCMoveAbsolute[mxMoveAbsNr].Velocity <> Velocity) THEN

	IF mxMoveAbsNr = 0 THEN
		mxMoveAbsNr :=1;
	ELSE
		mxMoveAbsNr :=0;
	END_IF
	
	(*Write parameters*)
	MCMoveAbsolute[mxMoveAbsNr].Position:=Position;
	MCMoveAbsolute[mxMoveAbsNr].Velocity:=Velocity;
(*	IF Velocity > 0.0 	THEN  MCMoveAbsolute[mxMoveAbsNr].Velocity:=Velocity; 		 ELSE MCMoveAbsolute[mxMoveAbsNr].Velocity:=parameters.VelocityAuto; 	END_IF*) 
END_IF

MCMoveAbsolute[mxMoveAbsNr].Execute:=TRUE;

(* Return value *)
M_MoveAbsolute:=MCMoveAbsolute[mxMoveAbsNr].Done;
END_METHOD

METHOD M_MoveVelocity : BOOL
VAR_INPUT
	Velocity			: LREAL;			
	Direction			: MC_Direction;
END_VAR
(*compare for different setpoints, if so change fb mcMoveVelocity*)
IF 	(MCMoveVelocity[mxMoveVelocityNr].Velocity <> Velocity) THEN

	IF mxMoveVelocityNr = 0 THEN
		mxMoveVelocityNr :=1;
	ELSE
		mxMoveVelocityNr :=0;
	END_IF

	(*Write parameters*)
	MCMoveVelocity[mxMoveVelocityNr].Velocity:=Velocity;
(*	IF Velocity > 0 	THEN MCMoveVelocity[mxMoveVelocityNr].Velocity:=Velocity; 			ELSE MCMoveVelocity[mxMoveVelocityNr].Velocity:=parameters.VelocityAuto; 		END_IF*)

END_IF

MCMoveVelocity[mxMoveVelocityNr].Execute:=TRUE;
MCMoveVelocity[mxMoveVelocityNr].Direction:=Direction;

(*Give return value*)
M_MoveVelocity:=MCMoveVelocity[mxMoveVelocityNr].Active;
END_METHOD

METHOD M_ReadParameter : LREAL
VAR_INPUT
		miParameterNr:INT;
END_VAR
MCReadParameter.ParameterNumber:=miParameterNr;
MCReadParameter.Enable:=TRUE;

M_ReadParameter:=MCReadParameter.Value;
END_METHOD

METHOD M_Reset : BOOL
VAR_INPUT
	
END_VAR

(* Return Value *)
M_Reset:= MCReset.Done;
END_METHOD

METHOD M_SetPosition : BOOL
VAR_INPUT
	NewPosition:LREAL;
END_VAR
MCSetPosition.Position:=NewPosition;
MCSetPosition.Execute:=TRUE;

M_SetPosition:=MCSetPosition.Done;
END_METHOD

METHOD M_Stop : BOOL
MCStop.Execute:=TRUE;

(* Return Value *)
M_Stop:= MCStop.Done;
END_METHOD

METHOD M_WriteParameter : BOOL
VAR_INPUT
	miParameterNr:INT;
	miValue:LREAL;
END_VAR
MCWriteParameter.ParameterNumber:=miParameterNr;
MCWriteParameter.Value:=miValue;
MCWriteParameter.Execute:=TRUE;

M_WriteParameter:=MCWriteParameter.Done;
END_METHOD

ACTION WritePosBias:
(*StateChange (Transition)  Signalgeneration*)
mxPosBiasTransitionState:=(miPosBiasState<>miPosBiasOldstate);
(*State text*)
sPosBiasStateText:=sPosBiasStateTextDef[miPosBiasState];
(*Timeout Watchdog for Statemachine*)
mxPosBiasTimeoutEnable:=NOT (miPosBiasState=0)  AND NOT mxReset;

PosBiasTimeout(IN:=mxPosBiasTimeoutEnable  , PT:=tPosBiasStateTimeouts[miPosBiasState] );
PosBiasTimeOutUpFlank(CLK:=PosBiasTimeout.Q );
miPosBiasOldstate:=miPosBiasState;

(*Set Errorbit when Raising edge of Timeout has been detected*)
IF PosBiasTimeOutUpFlank.Q THEN
	exPosBiasTimeOut:=TRUE; 			(* 1 Timeout for the whole programcycle *)
END_IF

(*Function to reset the Statemachine*)
IF mxResetPosBiasState THEN
	mxResetPosBiasState:=FALSE;
	miPosBiasState:=0;
	miPosBiasOldstate:=miPosBiasState;
	mxPosBiasTransitionState:=FALSE;

	AdsReadPosBias.READ:= FALSE;
	AdsWritePosBias.WRITE:= FALSE;

	mxZeroCommand:= FALSE;
	SignalLightStatus:= FALSE;
END_IF

AdsReadPosBias(
	NETID:= '',
	PORT:= 500,
	IDXGRP:= SysParameters.IDXGRP,
	IDXOFFS:= 16#7,
	LEN:= 8,
	DESTADDR:= ADR(PositionBiasRead),
	TMOUT:= T#1s);

AdsWritePosBias(
	NETID:= '',
	PORT:= 500,
	IDXGRP:= SysParameters.IDXGRP,
	IDXOFFS:= 16#7,
	LEN:= 8,
	SRCADDR:= ADR(SysParameters.PositionBias),
	TMOUT:= T#1s);

(*Definition State has Error*)
mxPosBiasHasError:=FALSE;

(*Cycle State's*)
CASE miPosBiasState OF
	(*Wait for Start *)
	0:
		(* Zero command from HMI *)
		IF mxZeroCommand THEN
			mxZeroCommand:= FALSE;
			SignalLightStatus:= FALSE;

			AdsReadPosBias.READ:= TRUE;
			miPosBiasState:= 1;
		END_IF

		(* PLC startup *)
		IF mxFirstCycle THEN
			SignalLightStatus:= FALSE;

			AdsWritePosBias.WRITE:= TRUE;
			miPosBiasState:= 2;
		END_IF

	(* Calculate new Position Bias with actual bias and act position *)
	1:
		IF NOT AdsReadPosBias.BUSY THEN
			AdsReadPosBias.READ:= FALSE;

			SysParameters.PositionBias:= mrHomePos - axAxis.NcToPlc.ActPos + PositionBiasRead;
			AdsWritePosBias.WRITE:= TRUE;

			miPosBiasState:= 2;
		END_IF

	(* Write new position bias *)
	2:
		IF NOT AdsWritePosBias.BUSY THEN
			AdsWritePosBias.WRITE:= FALSE;
			SignalLightStatus:= TRUE;

			miPosBiasState:= 0;
		END_IF
END_CASE

(*Set Busy bit FOR Statemachine*)
mxPosBiasBusy:=(miposBiasState<>0);
END_ACTION

END_FUNCTION_BLOCK

// ---- POUs/InMoldDrying/TransferMold/FB_TransferMold.TcPOU
FUNCTION_BLOCK FB_TransferMold
VAR CONSTANT
	sCycleStateTextDef: ARRAY[0..25]  OF STRING :=	
		['State 0: Wait for Start',
		'State 1: Wait for product forming ready',
		'State 2: Move down',
		'State 3: Wait for move up signal from main cycle',
		'State 4: Move up with product, signal bottommold when free to move',
		'State 5: Wait for bottommold A or B is at IN position',
		'State 6: Move down tranfer to bottommold transfer position',
		'State 7: Transfer time (closed on bottommold)',
		'State 8: Move up with blowoff and stop blowoff at tranfermold position',
		'State 9: Wait for bottommold is out',
		'State 10: ',
		'State 11: ',
		'State 12: ',
		'State 13:',
		'State 14:',
		'State 15:',
		'State 16:',
		'State 17:',
		'State 18:',
		'State 19:',
		'State 20: [Pausing] Stop al hydraulic movement',
		'State 21: [Pausing] Move transfermold to up pause position',
		'State 22: [Paused] Wait for start',
		'State 23:',
		'State 24:',
		'State 25: Stop direct'];
	
	tCycleStateTimeouts: ARRAY[0..25] OF TIME := 
		[T#600S, 	// State 0:  Wait for Start
		T#5S,		// State 1:  Wait for product forming ready
		T#5S,		// State 2:  Move down
		T#5S,		// State 3:  Wait for move up signal from main cycle
		T#5S,		// State 4:  Move up with product, signal bottommold when free to move
		T#5S,		// State 5:  Wait for bottommold A or B is at IN position
		T#5S,		// State 6:  Move down tranfer to bottommold transfer position
		T#5S,		// State 7:  Transfer time (closed on bottommold)
		T#5S,		// State 8:  Move up with blowoff and stop blowoff at tranfermold position
		T#5S,		// State 9:  Wait for bottommold is out
		T#5S,		// State 10: 
		T#5S,		// State 11: 
		T#5S,		// State 12: 
		T#5S,		// State 13: 
		T#5S,		// State 14: 
		T#5S,		// State 15: 
		T#5S,		// State 16: 
		T#5S,		// State 17: 
		T#5S,		// State 18: 
		T#5S,		// State 19: 
		T#5S,		// State 20: [Pausing] Stop al hydraulic movement 
		T#5S,		// State 21: [Pausing] Move transfermold to up pause position
		T#5S,		// State 22: [Paused] Wait for start
		T#5S,		// State 23: 
		T#5S,		// State 24: 
		T#5S];		// State 25: Stop direct

	sInitStateTextDef: ARRAY[0..10] OF STRING :=
		['State 0: Wait for Init Start',
		'State 1: Move transfermold to up position',
		'State 2: Description Init State 2',
		'State 3: Description Init State 3',
		'State 4: Description Init State 4',
		'State 5: Description Init State 5',
		'State 6: Description Init State 6',
		'State 7: Description Init State 7',
		'State 8: Description Init State 8',
		'State 9: Description Init State 9',
		'State 10: Stop init state'];

	tInitStateTimeouts: ARRAY[0..10] OF TIME := 
		[T#10S,T#10S,T#10S,T#10S,T#10S,T#10S,T#10S,T#10S,T#10S,T#10S
		,T#10S];
END_VAR

VAR_INPUT
	mxReset							: BOOL;	(*Reset Error*)
	mxEmergency						: BOOL;
	mxAutoMode						: BOOL; (* TRUE = Automode *)
	mxEmptyMachine					: BOOL;

	mxResetCycleState				: BOOL;
	mxResetInitState				: BOOL;
	
	mxStartVacuum					: BOOL; (* Signal from product forming *)

	mxStartProductForming			: BOOL;
	RHSR_Blocked 					: BOOL;

	(*Singals.*)
	sgMoveUp						: BOOL; (* Signal from product forming *)
	sgMoveToTransferPosA			: BOOL;
	sgMoveToTransferPosB			: BOOL;
	sgMoveDownToFormingPos			: BOOL; (* Signal from product forming *)
	sgTrAtFormingPos				: BOOL; (* Signal to Product Forming, that transfer is down*)
	sgTrReleaseBmMoveIn				: BOOL; (* Signal to bottommold, is up, move in  *)
	sgTransferIsUpMoveOut			: BOOL; (* Signal to bottommold, is up, move out *)
	sgBottomMoldAIsOut				: BOOL;
	sgBottomMoldBIsOut				: BOOL;
	sgSample: BOOL;
END_VAR
VAR_IN_OUT
	ProdParameters					: ST_TransferMoldProdPar;
	MachParameters					: ST_TransferMoldMachPar;
END_VAR
VAR_OUTPUT
(*Errors*)
	Errors							: ST_TransferMoldErrors;
	mxErrorInit						: BOOL;		(* Error, stop immediately. Initialisation neccesary *)
	mxErrorStopinPos				: BOOL;		(* Error, stop in position. Only reset neccesary *)

(* State vars *)
	mxCycleBusy						: BOOL;
	mxInitBusy						: BOOL;
	
(* Vars *)
	mxInitialized					: BOOL;
	
	mxCilIsMovingIn					: BOOL;
	mxCilIsMovingOut				: BOOL;
	mxCilIsIn						: BOOL;
	mxCilIsOut						: BOOL;	

	DownPosition					: REAL; // Position at which the transfermold thinks its down.
	ActualPosition					: REAL;
	
	mxTransferIsUpMoveOutA			: BOOL; (* Signal to bottom Mold, move out *)
	mxTransferIsUpMoveOutB			: BOOL; (* Signal to bottom Mold, move out *)

	TransferPosA					: REAL;
	TransferPosB					: REAL;
END_VAR
VAR
(* State vars *)
	miCycleState					: INT :=0;
	miCycleOldstate					: INT :=0;
	mxCycleTransitionState			: BOOL := FALSE;
	sCycleStateText					: STRING;
	exCycleTimeOut					: BOOL;		(* Timeout for the whole programcycle *)
	CycleTimeout					: TON;
	CycleTimeOutUpFlank				: R_TRIG;
	mxCycleTimeoutEnable			: BOOL;
	CycleTime						: REAL;
	mxCycleHasError					: BOOL;
	miStopState						: INT;
	mxStartCycle					: BOOL;
	mxStopCycle						: BOOL;
	mxStopDirect					: BOOL;
	
	miInitState						: INT	:=0;
	miInitOldstate					: INT	:=0;
	mxInitTransitionState			: BOOL	:= FALSE;
	sInitStateText					: STRING;
	exInitTimeOut					: BOOL;		(* Timeout for the whole programcycle *)
	InitTimeout						: TON;
	InitTimeOutUpFlank				: R_TRIG;
	mxInitTimeoutEnable				: BOOL;
	InitTime						: REAL;
	mxInitHasError					: BOOL;
	mxStartInit						: BOOL;
	mxStopInit						: BOOL;
	

(* Objects *)
	HydraulicCilinder				: FB_HydraulicCilinderAnalog; (* Up, Down, Slow, Position *)
	Vacuum							: FB_MonoValveNoFdbck;	(* IMD-Y-082 *)		
	BlowOff							: FB_MonoValveNoFdbck;	(* IMD-Y-076 *)

(* Vars *)
	T_TransferTimeClosed			: TON;
	T_BlowOff						: TON;

	mxTransferToA					: BOOL;
	mxTransferToB					: BOOL;
	T_FormingTime					: TON;
	RT_StartForming					: R_TRIG;
	
	PositionHighSlow				: REAL;
	InitSlowPosition				: REAL;
	T_PauseDelayedUp: TON;
	mxInPause						: BOOL;
	T_TrToBmTimeout: TON;
	SR_TrDidNotReachTransferPos: SR;
	SR_TrDidNotReachFormingPos: SR;
	T_TrToFormTimeOut: TON;
	RT_TakeSample: R_TRIG;
END_VAR

Error();
Init();
Cycle();
Objects();

ActualPosition := HydraulicCilinder.ActPosition;
DownPosition := ProdParameters.PositionDownStop;

TransferPosA := ProdParameters.PositionTransferStopA;
TransferPosB := ProdParameters.PositionTransferStopB;

ACTION Cycle:
(*StateChange (Transition)  Signalgeneration*)
mxCycleTransitionState:=(miCycleState<>miCycleOldstate);
(*State text*)
sCycleStateText:=sCycleStateTextDef[miCycleState];
(*Timeout Watchdog for Statemachine*)
mxCycleTimeoutEnable:=NOT (miCycleState=0) AND NOT mxReset;

CycleTimeout(IN:=mxCycleTimeoutEnable, PT:=tCycleStateTimeouts[miCycleState] );
CycleTimeOutUpFlank(CLK:=CycleTimeout.Q );
miCycleOldstate:=miCycleState;

(*Set Errorbit when Raising edge of Timeout has been detected*)
IF CycleTimeOutUpFlank.Q THEN
	exCycleTimeOut:=TRUE; 			(* 1 Timeout for the whole programcycle *)
END_IF

(*Function to reset the Statemachine*)
IF mxResetCycleState THEN
	mxResetCycleState:= FALSE;
	mxInitialized := FALSE;
	
	miCycleState:=0;
	miCycleOldstate:=miCycleState;
	mxCycleTransitionState:=FALSE;

	T_TransferTimeClosed.IN:= FALSE;
	T_BlowOff.IN:= FALSE;
	sgTrReleaseBmMoveIn:= FALSE;
	sgTrAtFormingPos:= FALSE;
	mxTransferToA:= FALSE;
	mxTransferToB:= FALSE;
	sgTrReleaseBmMoveIn := FALSE;
	sgMoveToTransferPosA := FALSE;
	sgMoveToTransferPosB := FALSE;	
	mxTransferIsUpMoveOutA := FALSE;
	mxTransferIsUpMoveOutB := FALSE;
	SgTransferIsUpMoveOut := FALSE;
	sgMoveDownToFormingPos := FALSE;
	 mxEmptyMachine :=FALSE;
	T_TrToBmTimeout.IN := FALSE;
	T_TrToFormTimeOut.IN:=FALSE;
	sgSample:=FALSE;		
	mxStartCycle:= FALSE;
	mxStopCycle:= FALSE;
	mxStopDirect:=FALSE;
	
	HydraulicCilinder.M_Stop();
END_IF

(*Definition State has Error*)
mxCycleHasError:=FALSE;

T_TransferTimeClosed(PT:= MachParameters.TransferTimeClosed);
T_PauseDelayedUp(PT:=T#300MS);
T_TrToBmTimeout(PT:=T#5S);
T_TrToFormTimeOut(PT:=T#7S);

// When moving up with product (Step 6), start forming at forming position parameter
RT_StartForming(CLK:=((HydraulicCilinder.ActPosition >= MachParameters.PositionStartFormingProcess)AND (miCycleState=4)));
RT_TakeSample(CLK:=sgSample);

IF RT_TakeSample.Q THEN	Vacuum.M_Off(); END_IF
IF T_BlowOff.Q THEN BlowOff.M_Off(); END_IF

{region "copy parameter set for pause position movement"}
	 MachParameters.PausePositionUpSlow := MachParameters.PositionUpSlow;	
	 MachParameters.PausePositionUpCreep := MachParameters.PositionUpCreep;	
{endregion}

(*Cycle State's*)
CASE miCycleState OF
	0:  //(P) Wait for start from IMD
		IF mxStopCycle THEN
			mxStopCycle:= FALSE;
			miStopState:= miCycleState;
			miCycleState:= 20;
		ELSIF mxStartCycle THEN
			mxStartCycle:= FALSE;	
			miCycleState:= 1;
		END_IF

	1:  //(P)  Wait for formming product ready
		 HydraulicCilinder.M_Move(EndPosition:=MachParameters.PositionUpStop, NormalSpeed:= MachParameters.UpNormalSpeed, // Use the move method to keep the transfermold in its "UpStop" Postion.
									SlowPosition:=MachParameters.PositionUpStop - MachParameters.PositionUpSlow, SlowSpeed:=MachParameters.UpSlowSpeed,
									CreepPosition:=MachParameters.PositionUpStop - MachParameters.PositionUpCreep, CreepSpeed:=MachParameters.UpCreepSpeed);
		IF mxStopDirect THEN
			mxStopDirect:= FALSE;
			miCycleState:=25;
		ELSIF mxStopCycle AND mxEmptyMachine THEN
			mxStopCycle:= FALSE;
			mxEmptyMachine:= FALSE;
			HydraulicCilinder.M_Stop();
			miCycleState:= 0;
		ELSIF mxStopCycle THEN
			mxStopCycle:= FALSE;
			miStopState:= miCycleState;
			miCycleState:= 20;
		ELSIF sgMoveDownToFormingPos THEN	// signal from the Main cycle
			sgMoveDownToFormingPos:= FALSE;
			miCycleState:=2;
		END_IF
	
	2:  //(NP) Move transfer down to forming and open vacuum valve at pos X
		T_TrToFormTimeOut.IN:=TRUE;	
	
		IF HydraulicCilinder.ActPosition < (ProdParameters.PositionDownStop + MachParameters.PosDownStartVacOffset) THEN
			Vacuum.M_On();
		END_IF
		IF mxStopDirect THEN
			mxStopDirect:= FALSE;
			miCycleState:= 25;
		ELSIF HydraulicCilinder.M_Move(EndPosition:=ProdParameters.PositionDownStop, NormalSpeed:= MachParameters.DownSpeed, 
										SlowPosition:=ProdParameters.PositionDownStop + MachParameters.PositionDownSlow, SlowSpeed:=MachParameters.DownSpeedSlow,
										CreepPosition:=ProdParameters.PositionDownStop + MachParameters.PositionDownCreep, CreepSpeed:=MachParameters.DownSpeedCreep) OR T_TrToFormTimeOut.Q THEN		
			sgTrAtFormingPos:= TRUE;
			T_TrToFormTimeOut.IN:=FALSE;	
			miCycleState:= 3;
		END_IF
	
	3:  //(NP) Wait for product move signal from main cycle
		IF mxStopDirect THEN
			mxStopDirect:= FALSE;
			miCycleState:= 25;
		ELSIF sgMoveUp THEN
			sgMoveUp:= FALSE;
			miCycleState:= 4;
		END_IF
	
	4:	//(NP) Move up with product and signal when bottommold is free to move.
		IF RT_StartForming.q THEN
			mxStartProductForming:= TRUE;
		END_IF
		IF HydraulicCilinder.ActPosition > (MachParameters.PositionUpStop - ProdParameters.ReleaseBmMovementOffset) THEN 
			sgTrReleaseBmMoveIn := TRUE;
		END_IF;
		IF mxStopDirect THEN
			mxStopDirect:= FALSE;
			miCycleState:= 25;
		ELSIF HydraulicCilinder.M_Move(EndPosition:=MachParameters.PositionUpStop, NormalSpeed:= MachParameters.UpNormalSpeed, 
											SlowPosition:=MachParameters.PositionUpStop - MachParameters.PositionUpSlow, SlowSpeed:=MachParameters.UpSlowSpeed,
											CreepPosition:=MachParameters.PositionUpStop - MachParameters.PositionUpCreep, CreepSpeed:=MachParameters.UpCreepSpeed) THEN
			miCycleState:= 5;
		END_IF
				
	5: 	//(P)  Wait for bottom mold A OR B is IN 
		 HydraulicCilinder.M_Move(EndPosition:=MachParameters.PositionUpStop, NormalSpeed:= MachParameters.UpNormalSpeed, 	// Use the move method to keep the transfermold in its "UpStop" Postion.
									SlowPosition:=MachParameters.PositionUpStop - MachParameters.PositionUpSlow, SlowSpeed:=MachParameters.UpSlowSpeed,
									CreepPosition:=MachParameters.PositionUpStop - MachParameters.PositionUpCreep, CreepSpeed:=MachParameters.UpCreepSpeed);
		IF mxStopDirect THEN
			mxStopDirect:= FALSE;
			miCycleState:= 25;
		ELSIF mxStopCycle THEN
			mxStopCycle:= FALSE;
			miStopState:= miCycleState;
			miCycleState:= 20;
		ELSIF sgMoveToTransferPosA OR sgMoveToTransferPosB THEN
			sgTrReleaseBmMoveIn := FALSE;
			mxStartProductForming:= FALSE;
			miCycleState:= 6;
		END_IF
			
	6:	//(NP) Move transfer mold down to transfer position and close vacuum valve at pos X
		T_TrToBmTimeout.In := TRUE;		
	
		IF (sgMoveToTransferPosA AND (HydraulicCilinder.ActPosition < (ProdParameters.PositionTransferStopA + MachParameters.PosTrStopVacOffset))) OR
 			(sgMoveToTransferPosB AND (HydraulicCilinder.ActPosition < (ProdParameters.PositionTransferStopB + MachParameters.PosTrStopVacOffset)))THEN
			Vacuum.M_Off();
		END_IF
		// Removed from step 9 at the request of mathijs wever:
		(*	Removed and moved Blowff.M_On to when the transfermold is closed on the bottommold. on the request of Matthijs Wever.
		IF (sgMoveToTransferPosA AND (HydraulicCilinder.ActPosition < ( ProdParameters.PositionTransferStopA + MachParameters.PosTrStartBlowOffOffset))) OR
			(sgMoveToTransferPosB AND (HydraulicCilinder.ActPosition < ( ProdParameters.PositionTransferStopB + MachParameters.PosTrStartBlowOffOffset))) THEN
			BlowOff.M_On();
		END_IF
		*)
		IF mxStopDirect THEN
			mxStopDirect:= FALSE;
			miCycleState:= 25;
		ELSIF sgMoveToTransferPosA THEN // A-Side mold.
			IF HydraulicCilinder.M_Move(EndPosition:=ProdParameters.PositionTransferStopA, NormalSpeed:= machParameters.DownSpeedToBm, 
										SlowPosition:=ProdParameters.PositionTransferStopA + MachParameters.PositionTransferSlow, machParameters.DownSpeedSlowToBm,
										CreepPosition:=ProdParameters.PositionTransferStopA + MachParameters.PositionTransferCreep, CreepSpeed:=machParameters.DownSpeedCreepToBm) OR T_TrToBmTimeout.Q THEN
				sgMoveToTransferPosA:= FALSE;
				mxTransferToA:= TRUE;
				mxTransferToB:= FALSE;
				BlowOff.M_On();			// BlowOff is now in this step, at the request of matthijs.
				T_TrToBmTimeout.In := FALSE;
				miCycleState:= 7;
			END_IF
		ELSIF sgMoveToTransferPosB THEN // B-side mold
			IF HydraulicCilinder.M_Move(EndPosition:=ProdParameters.PositionTransferStopB, NormalSpeed:= machParameters.DownSpeedToBm, 
										SlowPosition:=ProdParameters.PositionTransferStopB + MachParameters.PositionTransferSlow, SlowSpeed:=machParameters.DownSpeedSlowToBm,
										CreepPosition:=ProdParameters.PositionTransferStopB + MachParameters.PositionTransferCreep, CreepSpeed:=machParameters.DownSpeedCreepToBm) OR T_TrToBmTimeout.Q THEN
				sgMoveToTransferPosB:= FALSE;
				mxTransferToA:= FALSE;
				mxTransferToB:= TRUE;
				BlowOff.M_On();			// BlowOff is now in this step, at the request of matthijs.
				T_TrToBmTimeout.In := FALSE;
				miCycleState:= 7;
			END_IF
		END_IF

	7:  //(NP) Transfertime, while being closed*)
		T_TransferTimeClosed.IN:= TRUE;
		IF mxStopDirect THEN
			mxStopDirect:= FALSE;
			miCycleState:= 25;
		ELSIF T_TransferTimeClosed.Q THEN
			BlowOff.M_Off();
			T_TransferTimeClosed.IN:= FALSE;
			miCycleState:= 8;
		END_IF
	
	8:  //(NP) Move up with blowoff and stop blowoff at pos x of transfer
		(* // moved by the request of Siem H and Matthijs Wever
		IF (mxTransferToA AND (HydraulicCilinder.ActPosition < ( ProdParameters.PositionTransferStopA + MachParameters.PosTrStopBlowOffOffset))) OR
			(mxTransferToB AND (HydraulicCilinder.ActPosition < ( ProdParameters.PositionTransferStopB + MachParameters.PosTrStopBlowOffOffset))) THEN
			BlowOff.M_Off();
		END_IF*)
		IF mxStopDirect THEN
			mxStopDirect:= FALSE;
			miCycleState:= 25;
		ELSIF HydraulicCilinder.M_Move(EndPosition:=MachParameters.PositionUpStop, NormalSpeed:= machParameters.UpNormalSpeedToBm, 
										SlowPosition:=MachParameters.PositionUpStop - MachParameters.PositionUpSlow, SlowSpeed:=machParameters.UpSlowSpeedToBm,
										CreepPosition:=MachParameters.PositionUpStop - MachParameters.PositionUpCreep, CreepSpeed:=machParameters.UpCreepSpeedToBm) THEN
			sgTransferIsUpMoveOut:= TRUE;	
			miCycleState:= 9;
		END_IF
	
	9:  //(P)  Wait for BottomMold is OUT 	
		 HydraulicCilinder.M_Move(EndPosition:=MachParameters.PositionUpStop, NormalSpeed:= MachParameters.UpNormalSpeed,  // Use the move method to keep the transfermold in its "UpStop" Postion.
									SlowPosition:=MachParameters.PositionUpStop - MachParameters.PositionUpSlow, SlowSpeed:=MachParameters.UpSlowSpeed,
									CreepPosition:=MachParameters.PositionUpStop - MachParameters.PositionUpCreep, CreepSpeed:=MachParameters.UpCreepSpeed);
		IF mxStopDirect THEN
			mxStopDirect:= FALSE;
			miCycleState:= 25;
		ELSIF mxStopCycle THEN
			mxStopCycle:= FALSE;
			miStopState:= miCycleState;
			miCycleState:= 20;
		ELSIF (mxTransferToA AND sgBottomMoldAIsOut) OR (mxTransferToB AND sgBottomMoldBIsOut) THEN
			sgBottomMoldAIsOut := FALSE;
			sgBottomMoldBIsOut := FALSE;
			miCycleState:= 1;
		END_IF
		
	20: //(NP) Pause step, stop all movement
		T_PauseDelayedUp.IN := TRUE;
		
		IF mxStopDirect THEN
			mxStopDirect:= FALSE;	
			miCycleState:= 25;
		ELSIF T_PauseDelayedUp.Q AND HydraulicCilinder.M_Stop() THEN		
			miCycleState:= 21;
		END_IF

	21: //(NP) Move up to pause position 
		IF mxStopDirect THEN
			mxStopDirect:= FALSE;
			miCycleState:= 25;
		ELSIF HydraulicCilinder.M_Move(EndPosition:=MachParameters.PausePositionUp, NormalSpeed:= MachParameters.UpSlowSpeed, 
											SlowPosition:=MachParameters.PausePositionUp - MachParameters.PausePositionUpSlow, SlowSpeed:=MachParameters.UpSlowSpeed,
											CreepPosition:=MachParameters.PausePositionUp - MachParameters.PausePositionUpCreep, CreepSpeed:=MachParameters.UpCreepSpeed) THEN
			miCycleState := 22;
		END_IF
		
	22: //(Paused) Await restart. 
		IF mxStopDirect THEN
			mxStopDirect:= FALSE;
			miCycleState:= 25;
		ELSIF mxStartCycle THEN
			IF HydraulicCilinder.M_Move(EndPosition:=MachParameters.PositionUpStop, NormalSpeed:= MachParameters.UpSlowSpeed, // Use the move method to keep the transfermold in its "UpStop" Postion.
									SlowPosition:=MachParameters.PositionUpStop - MachParameters.PositionUpSlow, SlowSpeed:=MachParameters.UpSlowSpeed,
									CreepPosition:=MachParameters.PositionUpStop - MachParameters.PositionUpCreep, CreepSpeed:=MachParameters.UpCreepSpeed) THEN
				mxStartCycle:= FALSE;
				sgSample:=FALSE;
				miCycleState:= miStopState;
			END_IF
		END_IF

	25: // Stop Direct 
		HydraulicCilinder.M_StopDirect();
		Vacuum.M_Off();
		BlowOff.M_Off();
		sgTrReleaseBmMoveIn:= FALSE;
		sgTrAtFormingPos:= FALSE;
		mxTransferToA:= FALSE;
		mxTransferToB:= FALSE;
		sgTrReleaseBmMoveIn := FALSE;
		sgMoveToTransferPosA := FALSE;
		sgMoveToTransferPosB := FALSE;	
		mxTransferIsUpMoveOutA := FALSE;
		mxTransferIsUpMoveOutB := FALSE;
		SgTransferIsUpMoveOut := FALSE;
		sgMoveDownToFormingPos := FALSE;
		mxStartCycle:= FALSE;
		mxStopCycle:= FALSE;
		mxStopDirect:=FALSE;
		T_TrToBmTimeout.In := FALSE;
		T_TrToFormTimeOut.IN:=FALSE;
		sgSample:=FALSE;
		mxInitialized := FALSE;
		miCycleState:= 0;

END_CASE

mxCycleBusy:= miCycleState <> 0 AND NOT (miCycleState= 22);
mxInPause := miCycleState=22;
END_ACTION

ACTION Error:
SR_TrDidNotReachTransferPos(SET1:=T_TrToBmTimeout.Q, RESET:= mxReset, Q1=>Errors.TrDidNotReachBMPosTimeOut );
SR_TrDidNotReachFormingPos(SET1:=T_TrToFormTimeOut.Q, RESET:=mxReset, Q1=>Errors.TrDidNotReachFormingPosTimeOut);

(**********************************************************************************************************)
mxErrorStopinPos:= Errors.TrDidNotReachBMPosTimeOut OR Errors.TrDidNotReachFormingPosTimeOut;
mxErrorInit:= HydraulicCilinder.mxErrorInit;
END_ACTION

ACTION Init:
(*StateChange (Transition)  Signalgeneration*)
mxInitTransitionState:=(miInitState<>miInitOldstate);
(*State text*)
sInitStateText:=sInitStateTextDef[miInitState];
(*Timeout Watchdog for Statemachine*)
mxInitTimeoutEnable:=NOT (miInitState=0)  AND NOT mxReset;

InitTimeout(IN:=mxInitTimeoutEnable  , PT:=tInitStateTimeouts[miInitState] );
InitTimeOutUpFlank(CLK:=InitTimeout.Q );
miInitOldstate:=miInitState;

(*Set Errorbit when Raising edge of Timeout has been detected*)
IF InitTimeOutUpFlank.Q THEN
	exInitTimeOut:=TRUE; 			(* 1 Timeout for the whole programcycle *)
END_IF

(*Function to reset the Statemachine*)
IF mxResetInitState THEN
	mxResetInitState:=FALSE;
	miInitState:=0;
	miInitOldstate:=miInitState;
	mxInitTransitionState:=FALSE;
	
	mxStartInit:= FALSE;
	mxStopInit:= FALSE;
END_IF

(*Definition State has Error*)
mxInitHasError:=FALSE;

PositionHighSlow := MachParameters.PositionUpStop + (MachParameters.PositionUpStop - MachParameters.PositionUpSlow);


(*Init State's*)
CASE miInitState OF
	0:
		IF mxStartInit THEN
			mxStartInit:= FALSE;

			mxInitialized:= FALSE;
	(* If product then not switch off ?? *)
			Vacuum.M_Off();
			BlowOff.M_Off();	
			
			miInitState:= 1;
		END_IF

	1:
		IF mxStopInit THEN
			mxStopInit:= FALSE;

			miInitState:= 2;
		END_IF
	
		// Above normal position
		IF HydraulicCilinder.ActPosition > MachParameters.PositionUpStop THEN
			IF HydraulicCilinder.M_Move(EndPosition:=MachParameters.PositionUpStop, NormalSpeed:= MachParameters.InitDownNormalSpeed, 
										SlowPosition:=MachParameters.PositionUpStop + MachParameters.PositionUpSlow, SlowSpeed:=MachParameters.InitDownSpeedSlow,
										CreepPosition:=MachParameters.PositionUpStop + MachParameters.PositionUpCreep, CreepSpeed:=MachParameters.InitDownSpeedCreep) THEN			
			mxInitialized:= TRUE;
			miInitState:= 0;
			END_IF
			
		// Below normal position
		ELSE
			IF HydraulicCilinder.M_Move(EndPosition:=MachParameters.PositionUpStop, NormalSpeed:= MachParameters.InitupNormalSpeed, 
							SlowPosition:=MachParameters.PositionUpStop - MachParameters.PositionUpSlow, SlowSpeed:=MachParameters.InitUpSlowSpeed,
							CreepPosition:=MachParameters.PositionUpStop - MachParameters.PositionUpCreep, CreepSpeed:=MachParameters.InitUpCreepSpeed) THEN
			mxInitialized:= TRUE;
			miInitState:= 0;
			END_IF
		END_IF

	2:
		HydraulicCilinder.M_Stop();

		mxStartInit:= FALSE;
		mxStopInit:= FALSE;
		mxInitialized:=FALSE;					

		miInitState:= 0;
	
END_CASE

mxInitBusy:= miInitState<>0;
END_ACTION

METHOD M_EmptyMachine

IF mxCycleBusy THEN
	mxEmptyMachine:= TRUE;	
END_IF
END_METHOD

METHOD M_StartCycle
IF NOT mxCycleBusy THEN
	mxStartCycle:= TRUE;	
	mxStopCycle:=False;
END_IF
END_METHOD

METHOD M_StartInit

IF NOT mxInitBusy THEN 
	mxStartInit:= TRUE; 
END_IF
END_METHOD

